C01814=1092.503,260.660,421.963,177.107,20.191,152.904
C01815=1092.509,260.908,421.935,177.110,20.194,152.904
C01816=1092.515,261.157,421.907,177.114,20.196,152.904
C01817=1092.520,261.405,421.880,177.117,20.198,152.904
C01818=1092.526,261.654,421.852,177.120,20.200,152.904
C01819=1092.533,261.902,421.825,177.122,20.202,152.904
C01820=1092.538,262.150,421.797,177.126,20.204,152.904
C01821=1092.547,262.515,421.756,177.131,20.208,152.904
C01822=1092.555,262.879,421.715,177.135,20.211,152.904
C01823=1092.563,263.243,421.675,177.139,20.215,152.904
C01824=1092.572,263.608,421.634,177.144,20.218,152.904
C01825=1092.577,263.856,421.606,177.147,20.220,152.903
C01826=1092.583,264.105,421.578,177.150,20.222,152.903
C01827=1092.589,264.353,421.550,177.153,20.224,152.903
C01828=1092.595,264.601,421.522,177.157,20.227,152.903
C01829=1092.601,264.849,421.494,177.159,20.229,152.903
C01830=1092.606,265.097,421.466,177.162,20.231,152.903
C01831=1092.612,265.346,421.438,177.165,20.233,152.903
C01832=1092.617,265.594,421.410,177.169,20.236,152.903
C01833=1092.623,265.843,421.381,177.172,20.239,152.903
C01834=1092.629,266.091,421.353,177.174,20.241,152.904
C01835=1092.635,266.340,421.325,177.177,20.243,152.903
C01836=1092.640,266.588,421.297,177.181,20.245,152.903
C01837=1092.645,266.836,421.269,177.184,20.248,152.903
C01838=1092.651,267.085,421.241,177.187,20.250,152.904
C01839=1092.656,267.333,421.213,177.189,20.252,152.903
C01840=1092.662,267.581,421.184,177.193,20.254,152.903
C01841=1092.668,267.829,421.157,177.196,20.257,152.904
C01842=1092.674,268.078,421.128,177.199,20.259,152.903
C01843=1092.679,268.326,421.100,177.202,20.261,152.903
C01844=1092.685,268.575,421.072,177.206,20.264,152.903
C01845=1092.690,268.823,421.044,177.208,20.266,152.904
C01846=1092.697,269.071,421.015,177.211,20.268,152.903
C01847=1092.702,269.319,420.987,177.214,20.271,152.903
C01848=1092.708,269.568,420.959,177.218,20.273,152.903
C01849=1092.714,269.817,420.930,177.221,20.276,152.904
C01850=1092.719,270.065,420.902,177.223,20.278,152.904
C01851=1092.725,270.313,420.873,177.226,20.280,152.903
C01852=1092.730,270.561,420.845,177.230,20.282,152.904
C01853=1092.736,270.810,420.816,177.233,20.285,152.904
C01854=1092.741,271.058,420.788,177.236,20.287,152.904
C01855=1092.748,271.306,420.759,177.239,20.290,152.904
C01856=1092.753,271.554,420.731,177.242,20.292,152.904
C01857=1092.759,271.803,420.703,177.245,20.294,152.904
C01858=1092.764,272.051,420.674,177.248,20.296,152.904
C01859=1092.770,272.300,420.646,177.251,20.299,152.904
C01860=1092.776,272.548,420.617,177.254,20.301,152.904
C01861=1092.781,272.796,420.589,177.257,20.304,152.904
C01862=1092.787,273.044,420.560,177.261,20.306,152.904
C01863=1092.792,273.293,420.532,177.263,20.308,152.904
C01864=1092.798,273.541,420.503,177.266,20.311,152.904
C01865=1092.804,273.790,420.474,177.269,20.313,152.904
C01866=1092.810,274.037,420.446,177.273,20.316,152.904
C01867=1092.815,274.286,420.417,177.276,20.318,152.904
C01868=1092.821,274.534,420.388,177.279,20.321,152.904
C01869=1092.826,274.782,420.360,177.282,20.323,152.904
C01870=1092.832,275.031,420.331,177.285,20.325,152.904
C01871=1092.837,275.279,420.302,177.288,20.327,152.904
C01872=1092.843,275.528,420.274,177.291,20.330,152.904
C01873=1092.852,275.895,420.231,177.296,20.333,152.904
C01874=1092.860,276.262,420.188,177.300,20.337,152.904
C01875=1092.868,276.628,420.146,177.304,20.340,152.904
C01876=1092.877,276.995,420.104,177.309,20.344,152.904
C01877=1092.882,277.244,420.074,177.313,20.346,152.904
C01878=1092.888,277.492,420.045,177.316,20.349,152.904
C01879=1092.894,277.740,420.017,177.319,20.352,152.904
C01880=1092.899,277.988,419.987,177.322,20.354,152.904
C01881=1092.905,278.237,419.958,177.325,20.357,152.904
C01882=1092.910,278.485,419.930,177.328,20.359,152.904
C01883=1092.916,278.733,419.901,177.331,20.361,152.904
C01884=1092.922,278.981,419.871,177.334,20.364,152.904
C01885=1092.927,279.230,419.843,177.337,20.366,152.904
C01886=1092.933,279.478,419.814,177.340,20.369,152.904
C01887=1092.939,279.726,419.784,177.343,20.371,152.905
C01888=1092.945,279.974,419.755,177.346,20.374,152.905
C01889=1092.950,280.223,419.727,177.350,20.376,152.905
C01890=1092.956,280.471,419.698,177.353,20.379,152.905
C01891=1092.962,280.719,419.668,177.356,20.381,152.905
C01892=1092.968,280.967,419.639,177.359,20.384,152.905
C01893=1092.973,281.215,419.610,177.361,20.386,152.905
C01894=1092.979,281.463,419.581,177.365,20.388,152.905
C01895=1092.984,281.712,419.552,177.368,20.391,152.905
C01896=1092.990,281.961,419.522,177.371,20.393,152.905
C01897=1092.995,282.208,419.494,177.374,20.396,152.905
C01898=1093.001,282.457,419.464,177.377,20.398,152.905
C01899=1093.007,282.705,419.435,177.380,20.401,152.905
C01900=1093.013,282.953,419.405,177.384,20.404,152.905
C01901=1093.017,283.201,419.376,177.387,20.407,152.905
C01902=1093.024,283.449,419.347,177.390,20.409,152.905
C01903=1093.029,283.697,419.317,177.393,20.412,152.905
C01904=1093.035,283.946,419.288,177.396,20.414,152.905
C01905=1093.040,284.193,419.259,177.399,20.417,152.905
C01906=1093.046,284.442,419.229,177.402,20.419,152.905
C01907=1093.051,284.690,419.200,177.405,20.421,152.906
C01908=1093.058,284.938,419.171,177.408,20.424,152.906
C01909=1093.063,285.187,419.141,177.411,20.426,152.906
C01910=1093.069,285.435,419.112,177.414,20.429,152.906
C01911=1093.074,285.683,419.083,177.417,20.432,152.906
C01912=1093.080,285.931,419.053,177.420,20.434,152.906
C01913=1093.085,286.180,419.024,177.424,20.437,152.906
C01914=1093.091,286.427,418.993,177.427,20.439,152.906
C01915=1093.097,286.675,418.964,177.430,20.442,152.906
C01916=1093.103,286.924,418.935,177.433,20.444,152.906
C01917=1093.108,287.172,418.905,177.436,20.447,152.906
C01918=1093.114,287.420,418.876,177.439,20.450,152.906
C01919=1093.120,287.668,418.847,177.442,20.452,152.906
C01920=1093.125,287.916,418.816,177.445,20.455,152.906
C01921=1093.131,288.164,418.787,177.449,20.457,152.906
C01922=1093.137,288.413,418.758,177.452,20.460,152.906
C01923=1093.143,288.661,418.728,177.455,20.462,152.907
C01924=1093.149,288.909,418.698,177.458,20.465,152.907
C01925=1093.157,289.285,418.653,177.463,20.469,152.907
C01926=1093.166,289.662,418.608,177.467,20.473,152.907
C01927=1093.174,290.038,418.562,177.472,20.477,152.907
C01928=1093.184,290.415,418.517,177.477,20.481,152.907
C01929=1093.188,290.663,418.488,177.480,20.484,152.907
C01930=1093.194,290.911,418.458,177.483,20.486,152.907
C01931=1093.200,291.159,418.428,177.486,20.489,152.907
C01932=1093.205,291.407,418.398,177.489,20.492,152.907
C01933=1093.211,291.655,418.368,177.492,20.494,152.907
C01934=1093.217,291.903,418.338,177.496,20.497,152.908
C01935=1093.222,292.151,418.308,177.498,20.500,152.908
C01936=1093.228,292.400,418.278,177.502,20.502,152.908
C01937=1093.234,292.648,418.248,177.505,20.505,152.908
C01938=1093.239,292.896,418.218,177.508,20.508,152.908
C01939=1093.245,293.144,418.188,177.511,20.510,152.908
C01940=1093.251,293.392,418.158,177.514,20.513,152.908
C01941=1093.256,293.640,418.128,177.517,20.516,152.908
C01942=1093.262,293.889,418.098,177.520,20.518,152.908
C01943=1093.268,294.136,418.068,177.523,20.521,152.908
C01944=1093.273,294.385,418.038,177.526,20.524,152.909
C01945=1093.279,294.633,418.008,177.530,20.526,152.909
C01946=1093.285,294.880,417.978,177.533,20.529,152.909
C01947=1093.290,295.129,417.948,177.536,20.532,152.909
C01948=1093.296,295.377,417.918,177.539,20.534,152.909
C01949=1093.302,295.625,417.887,177.542,20.537,152.909
C01950=1093.308,295.873,417.858,177.545,20.540,152.909
C01951=1093.313,296.121,417.827,177.548,20.542,152.909
C01952=1093.319,296.369,417.797,177.551,20.545,152.909
C01953=1093.325,296.616,417.767,177.554,20.548,152.909
C01954=1093.330,296.865,417.737,177.557,20.550,152.909
C01955=1093.336,297.113,417.706,177.560,20.553,152.910
C01956=1093.341,297.361,417.676,177.564,20.556,152.910
C01957=1093.348,297.609,417.645,177.567,20.559,152.910
C01958=1093.353,297.858,417.615,177.570,20.561,152.910
C01959=1093.359,298.106,417.585,177.573,20.564,152.910
C01960=1093.364,298.354,417.554,177.576,20.567,152.910
C01961=1093.370,298.602,417.524,177.579,20.570,152.910
C01962=1093.376,298.849,417.493,177.582,20.572,152.910
C01963=1093.381,299.098,417.462,177.585,20.575,152.911
C01964=1093.386,299.346,417.433,177.588,20.578,152.911
C01965=1093.392,299.594,417.402,177.592,20.581,152.911
C01966=1093.397,299.842,417.371,177.595,20.584,152.911
C01967=1093.403,300.090,417.341,177.598,20.587,152.911
C01968=1093.409,300.338,417.311,177.601,20.590,152.911
C01969=1093.414,300.586,417.280,177.604,20.593,152.911
C01970=1093.420,300.834,417.249,177.607,20.596,152.912
C01971=1093.425,301.082,417.218,177.610,20.598,152.912
C01972=1093.431,301.330,417.188,177.613,20.601,152.912
C01973=1093.437,301.578,417.157,177.616,20.604,152.912
C01974=1093.442,301.826,417.126,177.619,20.607,152.912
C01975=1093.448,302.074,417.096,177.622,20.609,152.912
C01976=1093.453,302.322,417.065,177.625,20.612,152.913
C01977=1093.463,302.712,417.017,177.631,20.617,152.913
C01978=1093.471,303.103,416.968,177.635,20.621,152.913
C01979=1093.480,303.493,416.920,177.640,20.626,152.913
C01980=1093.489,303.884,416.871,177.645,20.630,152.913
C01981=1093.495,304.131,416.841,177.648,20.633,152.914
C01982=1093.500,304.380,416.810,177.651,20.636,152.914
C01983=1093.506,304.627,416.779,177.655,20.639,152.914
C01984=1093.512,304.876,416.747,177.658,20.642,152.914
C01985=1093.517,305.123,416.717,177.661,20.645,152.914
C01986=1093.523,305.372,416.686,177.664,20.648,152.914
C01987=1093.528,305.619,416.656,177.667,20.651,152.914
C01988=1093.534,305.867,416.624,177.670,20.654,152.915
C01989=1093.540,306.115,416.593,177.673,20.657,152.915
C01990=1093.545,306.364,416.562,177.676,20.659,152.915
C01991=1093.551,306.611,416.531,177.679,20.662,152.915
C01992=1093.556,306.859,416.500,177.683,20.666,152.915
C01993=1093.563,307.107,416.470,177.686,20.669,152.915
C01994=1093.568,307.355,416.438,177.689,20.672,152.916
C01995=1093.574,307.603,416.408,177.692,20.674,152.916
C01996=1093.580,307.852,416.376,177.695,20.677,152.916
C01997=1093.586,308.099,416.345,177.698,20.680,152.916
C01998=1093.591,308.347,416.314,177.701,20.683,152.916
C01999=1093.597,308.594,416.283,177.705,20.686,152.916
C02000=1093.603,308.843,416.252,177.708,20.689,152.916
C02001=1093.608,309.090,416.220,177.711,20.692,152.917
C02002=1093.614,309.338,416.190,177.714,20.695,152.917
C02003=1093.620,309.586,416.158,177.717,20.698,152.917
C02004=1093.626,309.834,416.128,177.720,20.701,152.917
C02005=1093.632,310.083,416.096,177.723,20.703,152.917
C02006=1093.637,310.331,416.065,177.726,20.706,152.917
C02007=1093.643,310.578,416.034,177.730,20.710,152.918
C02008=1093.649,310.827,416.002,177.733,20.713,152.918
C02009=1093.655,311.074,415.971,177.735,20.716,152.918
C02010=1093.660,311.323,415.940,177.738,20.719,152.918
C02011=1093.666,311.570,415.908,177.742,20.721,152.918
C02012=1093.672,311.817,415.877,177.745,20.724,152.918
C02013=1093.678,312.066,415.846,177.748,20.728,152.919
C02014=1093.683,312.314,415.814,177.751,20.731,152.919
C02015=1093.690,312.562,415.783,177.754,20.734,152.919
C02016=1093.695,312.810,415.752,177.757,20.737,152.919
C02017=1093.701,313.058,415.720,177.760,20.740,152.919
C02018=1093.707,313.305,415.689,177.763,20.743,152.920
C02019=1093.713,313.554,415.657,177.766,20.746,152.920
C02020=1093.718,313.802,415.626,177.770,20.749,152.920
C02021=1093.724,314.050,415.594,177.773,20.751,152.920
C02022=1093.730,314.297,415.563,177.776,20.754,152.920
C02023=1093.736,314.546,415.531,177.779,20.757,152.920
C02024=1093.741,314.793,415.500,177.782,20.760,152.921
C02025=1093.748,315.041,415.468,177.786,20.764,152.921
C02026=1093.753,315.289,415.437,177.789,20.767,152.921
C02027=1093.759,315.537,415.405,177.792,20.770,152.921
C02028=1093.765,315.784,415.373,177.795,20.773,152.922
C02029=1093.773,316.178,415.322,177.800,20.778,152.922
C02030=1093.782,316.571,415.272,177.804,20.783,152.922
C02031=1093.791,316.964,415.222,177.809,20.788,152.923
C02032=1093.799,317.357,415.171,177.814,20.793,152.923
C02033=1093.805,317.605,415.139,177.817,20.797,152.923
C02034=1093.811,317.853,415.108,177.820,20.800,152.924
C02035=1093.817,318.101,415.076,177.823,20.803,152.924
C02036=1093.822,318.349,415.044,177.827,20.807,152.924
C02037=1093.828,318.597,415.012,177.830,20.810,152.924
C02038=1093.833,318.844,414.980,177.833,20.813,152.924
C02039=1093.839,319.093,414.948,177.835,20.816,152.925
C02040=1093.845,319.340,414.916,177.838,20.819,152.925
C02041=1093.850,319.589,414.884,177.842,20.822,152.925
C02042=1093.855,319.836,414.852,177.845,20.826,152.926
C02043=1093.861,320.084,414.820,177.848,20.829,152.926
C02044=1093.867,320.333,414.788,177.851,20.832,152.926
C02045=1093.873,320.579,414.756,177.855,20.836,152.926
C02046=1093.879,320.828,414.724,177.858,20.839,152.926
C02047=1093.884,321.075,414.691,177.860,20.842,152.927
C02048=1093.890,321.324,414.659,177.863,20.845,152.927
C02049=1093.895,321.571,414.628,177.867,20.849,152.927
C02050=1093.901,321.819,414.595,177.870,20.852,152.927
C02051=1093.907,322.067,414.563,177.873,20.855,152.928
C02052=1093.913,322.315,414.531,177.876,20.858,152.928
C02053=1093.918,322.563,414.499,177.879,20.862,152.928
C02054=1093.924,322.811,414.466,177.882,20.865,152.929
C02055=1093.930,323.058,414.434,177.885,20.868,152.929
C02056=1093.936,323.306,414.402,177.888,20.872,152.929
C02057=1093.941,323.555,414.370,177.892,20.875,152.929
C02058=1093.946,323.802,414.337,177.894,20.878,152.930
C02059=1093.952,324.050,414.305,177.897,20.881,152.930
C02060=1093.958,324.298,414.273,177.900,20.885,152.930
C02061=1093.963,324.545,414.240,177.904,20.888,152.930
C02062=1093.969,324.794,414.208,177.907,20.892,152.931
C02063=1093.976,325.041,414.176,177.910,20.895,152.931
C02064=1093.981,325.289,414.144,177.912,20.898,152.931
C02065=1093.986,325.537,414.111,177.916,20.902,152.932
C02066=1093.993,325.785,414.078,177.919,20.905,152.932
C02067=1093.999,326.033,414.046,177.922,20.908,152.932
C02068=1094.004,326.280,414.014,177.926,20.912,152.932
C02069=1094.010,326.528,413.981,177.928,20.915,152.933
C02070=1094.016,326.776,413.949,177.931,20.918,152.933
C02071=1094.022,327.024,413.917,177.934,20.921,152.933
C02072=1094.027,327.272,413.883,177.938,20.925,152.933
C02073=1094.033,327.519,413.851,177.941,20.928,152.934
C02074=1094.039,327.767,413.819,177.944,20.932,152.934
C02075=1094.045,328.015,413.786,177.947,20.936,152.934
C02076=1094.051,328.263,413.754,177.950,20.939,152.935
C02077=1094.057,328.511,413.721,177.953,20.942,152.935
C02078=1094.062,328.758,413.688,177.956,20.946,152.935
C02079=1094.068,329.006,413.656,177.959,20.949,152.935
C02080=1094.074,329.254,413.623,177.962,20.952,152.936
C02081=1094.083,329.640,413.572,177.967,20.958,152.936
C02082=1094.092,330.027,413.521,177.972,20.963,152.937
C02083=1094.101,330.413,413.470,177.977,20.969,152.937
C02084=1094.110,330.799,413.419,177.982,20.974,152.938
C02085=1094.116,331.046,413.386,177.985,20.978,152.938
C02086=1094.122,331.295,413.354,177.988,20.981,152.938
C02087=1094.128,331.543,413.320,177.991,20.984,152.939
C02088=1094.134,331.790,413.288,177.995,20.988,152.939
C02089=1094.140,332.038,413.254,177.997,20.991,152.939
C02090=1094.145,332.285,413.222,178.000,20.995,152.940
C02091=1094.151,332.533,413.189,178.004,20.999,152.940
C02092=1094.156,332.781,413.155,178.006,21.002,152.940
C02093=1094.162,333.029,413.123,178.009,21.005,152.941
C02094=1094.168,333.277,413.090,178.013,21.009,152.941
C02095=1094.173,333.525,413.057,178.016,21.013,152.941
C02096=1094.180,333.772,413.024,178.019,21.017,152.942
C02097=1094.185,334.020,412.991,178.022,21.020,152.942
C02098=1094.190,334.267,412.958,178.025,21.023,152.942
C02099=1094.197,334.515,412.925,178.028,21.027,152.943
C02100=1094.202,334.763,412.891,178.031,21.031,152.943
C02101=1094.208,335.011,412.858,178.035,21.035,152.943
C02102=1094.213,335.259,412.825,178.037,21.039,152.944
C02103=1094.220,335.506,412.792,178.040,21.042,152.944
C02104=1094.225,335.754,412.759,178.044,21.046,152.944
C02105=1094.231,336.002,412.725,178.047,21.049,152.945
C02106=1094.237,336.249,412.692,178.050,21.053,152.945
C02107=1094.243,336.497,412.659,178.053,21.057,152.945
C02108=1094.248,336.745,412.625,178.055,21.060,152.946
C02109=1094.254,336.993,412.592,178.059,21.064,152.946
C02110=1094.260,337.240,412.559,178.062,21.068,152.947
C02111=1094.266,337.488,412.526,178.066,21.072,152.947
C02112=1094.272,337.736,412.492,178.068,21.075,152.947
C02113=1094.277,337.984,412.458,178.071,21.079,152.948
C02114=1094.283,338.231,412.425,178.074,21.083,152.948
C02115=1094.289,338.479,412.392,178.077,21.086,152.948
C02116=1094.295,338.727,412.359,178.081,21.090,152.949
C02117=1094.300,338.974,412.325,178.083,21.094,152.949
C02118=1094.306,339.222,412.292,178.087,21.098,152.950
C02119=1094.312,339.470,412.258,178.090,21.102,152.950
C02120=1094.317,339.717,412.224,178.093,21.105,152.950
C02121=1094.323,339.965,412.191,178.096,21.109,152.951
C02122=1094.329,340.213,412.158,178.099,21.113,152.951
C02123=1094.334,340.460,412.124,178.102,21.117,152.952
C02124=1094.340,340.708,412.090,178.105,21.120,152.952
C02125=1094.346,340.956,412.056,178.108,21.125,152.953
C02126=1094.351,341.204,412.023,178.111,21.128,152.953
C02127=1094.357,341.451,411.989,178.114,21.133,152.953
C02128=1094.363,341.699,411.955,178.117,21.136,152.954
C02129=1094.368,341.947,411.922,178.121,21.140,152.954
C02130=1094.375,342.195,411.888,178.123,21.144,152.955
C02131=1094.380,342.443,411.854,178.127,21.148,152.955
C02132=1094.386,342.690,411.820,178.129,21.152,152.955
C02133=1094.395,343.070,411.769,178.134,21.158,152.956
C02134=1094.404,343.450,411.717,178.139,21.164,152.957
C02135=1094.413,343.830,411.664,178.144,21.170,152.957
C02136=1094.421,344.210,411.613,178.149,21.176,152.958
C02137=1094.428,344.458,411.579,178.151,21.179,152.958
C02138=1094.433,344.706,411.546,178.155,21.184,152.959
C02139=1094.439,344.953,411.511,178.157,21.187,152.959
C02140=1094.445,345.200,411.477,178.161,21.192,152.960
C02141=1094.450,345.449,411.444,178.163,21.196,152.960
C02142=1094.456,345.696,411.409,178.167,21.200,152.961
C02143=1094.462,345.944,411.375,178.170,21.203,152.961
C02144=1094.468,346.191,411.341,178.173,21.208,152.962
C02145=1094.474,346.439,411.308,178.176,21.212,152.962
C02146=1094.479,346.687,411.273,178.179,21.216,152.963
C02147=1094.485,346.934,411.239,178.183,21.220,152.963
C02148=1094.491,347.181,411.205,178.185,21.224,152.964
C02149=1094.497,347.429,411.170,178.189,21.228,152.964
C02150=1094.502,347.677,411.137,178.191,21.232,152.965
C02151=1094.508,347.925,411.102,178.195,21.237,152.965
C02152=1094.514,348.172,411.068,178.197,21.240,152.965
C02153=1094.520,348.420,411.034,178.201,21.245,152.966
C02154=1094.525,348.668,410.999,178.203,21.249,152.966
C02155=1094.531,348.915,410.965,178.207,21.253,152.967
C02156=1094.537,349.162,410.931,178.210,21.257,152.967
C02157=1094.542,349.410,410.897,178.213,21.261,152.968
C02158=1094.549,349.658,410.862,178.216,21.265,152.968
C02159=1094.554,349.905,410.828,178.219,21.269,152.969
C02160=1094.559,350.153,410.793,178.222,21.274,152.969
C02161=1094.566,350.401,410.759,178.224,21.278,152.970
C02162=1094.572,350.648,410.725,178.228,21.282,152.970
C02163=1094.577,350.896,410.690,178.231,21.286,152.971
C02164=1094.583,351.143,410.656,178.234,21.290,152.971
C02165=1094.589,351.391,410.622,178.237,21.295,152.972
C02166=1094.594,351.638,410.587,178.240,21.299,152.972
C02167=1094.600,351.886,410.553,178.243,21.303,152.973
C02168=1094.606,352.133,410.517,178.247,21.308,152.973
C02169=1094.612,352.381,410.483,178.249,21.311,152.974
C02170=1094.618,352.628,410.449,178.252,21.316,152.975
C02171=1094.624,352.876,410.414,178.255,21.320,152.975
C02172=1094.630,353.123,410.380,178.258,21.324,152.976
C02173=1094.635,353.370,410.345,178.262,21.329,152.976
C02174=1094.641,353.618,410.311,178.264,21.333,152.977
C02175=1094.647,353.866,410.276,178.268,21.338,152.977
C02176=1094.652,354.113,410.242,178.271,21.342,152.978
C02177=1094.658,354.361,410.206,178.273,21.346,152.978
C02178=1094.664,354.608,410.172,178.277,21.351,152.979
C02179=1094.669,354.856,410.137,178.279,21.355,152.979
C02180=1094.675,355.104,410.102,178.283,21.359,152.980
C02181=1094.681,355.351,410.068,178.286,21.364,152.981
C02182=1094.686,355.598,410.033,178.288,21.368,152.981
C02183=1094.693,355.846,409.998,178.292,21.372,152.982
C02184=1094.698,356.093,409.963,178.295,21.377,152.982
C02185=1094.708,356.476,409.909,178.299,21.384,152.983
C02186=1094.716,356.858,409.855,178.304,21.391,152.984
C02187=1094.726,357.242,409.801,178.308,21.398,152.985
C02188=1094.734,357.624,409.747,178.314,21.405,152.986
C02189=1094.740,357.871,409.712,178.316,21.409,152.986
C02190=1094.745,358.119,409.677,178.319,21.414,152.987
C02191=1094.752,358.366,409.642,178.323,21.418,152.988
C02192=1094.758,358.614,409.607,178.325,21.422,152.988
C02193=1094.763,358.861,409.572,178.328,21.427,152.989
C02194=1094.770,359.108,409.537,178.332,21.432,152.989
C02195=1094.775,359.356,409.502,178.334,21.436,152.990
C02196=1094.781,359.604,409.466,178.337,21.441,152.991
C02197=1094.787,359.850,409.432,178.341,21.446,152.991
C02198=1094.793,360.099,409.397,178.344,21.450,152.992
C02199=1094.798,360.346,409.361,178.346,21.454,152.992
C02200=1094.804,360.593,409.326,178.350,21.459,152.993
C02201=1094.810,360.840,409.291,178.353,21.464,152.994
C02202=1094.816,361.088,409.256,178.355,21.468,152.994
C02203=1094.821,361.335,409.220,178.358,21.473,152.995
C02204=1094.827,361.583,409.185,178.362,21.478,152.996
C02205=1094.833,361.830,409.149,178.365,21.483,152.996
C02206=1094.839,362.078,409.114,178.367,21.487,152.997
C02207=1094.845,362.325,409.080,178.371,21.492,152.998
C02208=1094.851,362.573,409.044,178.374,21.497,152.998
C02209=1094.856,362.820,409.008,178.377,21.502,152.999
C02210=1094.862,363.067,408.973,178.379,21.506,153.000
C02211=1094.868,363.315,408.937,178.383,21.511,153.000
C02212=1094.874,363.562,408.902,178.386,21.516,153.001
C02213=1094.880,363.810,408.866,178.389,21.521,153.002
C02214=1094.885,364.057,408.831,178.391,21.525,153.002
C02215=1094.891,364.304,408.795,178.394,21.530,153.003
C02216=1094.897,364.551,408.759,178.398,21.535,153.004
C02217=1094.903,364.799,408.724,178.401,21.540,153.004
C02218=1094.909,365.046,408.689,178.403,21.544,153.005
C02219=1094.915,365.293,408.653,178.406,21.549,153.006
C02220=1094.921,365.541,408.617,178.409,21.554,153.006
C02221=1094.926,365.788,408.582,178.413,21.559,153.007
C02222=1094.932,366.035,408.546,178.416,21.564,153.008
C02223=1094.938,366.283,408.511,178.418,21.569,153.008
C02224=1094.943,366.530,408.475,178.421,21.574,153.009
C02225=1094.949,366.778,408.438,178.424,21.579,153.010
C02226=1094.955,367.024,408.403,178.427,21.584,153.011
C02227=1094.961,367.272,408.367,178.431,21.589,153.011
C02228=1094.967,367.520,408.331,178.433,21.593,153.012
C02229=1094.972,367.767,408.296,178.436,21.599,153.013
C02230=1094.979,368.014,408.260,178.439,21.604,153.013
C02231=1094.984,368.262,408.223,178.442,21.609,153.014
C02232=1094.989,368.509,408.188,178.445,21.614,153.015
C02233=1094.995,368.756,408.152,178.448,21.619,153.016
C02234=1095.001,369.003,408.116,178.451,21.623,153.016
C02235=1095.007,369.251,408.080,178.454,21.629,153.017
C02236=1095.013,369.498,408.045,178.457,21.634,153.018
C02237=1095.022,369.896,407.986,178.462,21.642,153.019
C02238=1095.032,370.294,407.928,178.467,21.650,153.020
C02239=1095.041,370.691,407.870,178.471,21.658,153.022
C02240=1095.050,371.089,407.813,178.475,21.667,153.023
C02241=1095.057,371.337,407.776,178.479,21.672,153.024
C02242=1095.061,371.584,407.740,178.482,21.677,153.024
C02243=1095.068,371.831,407.704,178.485,21.682,153.025
C02244=1095.074,372.079,407.668,178.488,21.687,153.026
C02245=1095.080,372.326,407.632,178.491,21.693,153.027
C02246=1095.085,372.572,407.595,178.494,21.698,153.028
C02247=1095.091,372.820,407.559,178.496,21.703,153.028
C02248=1095.097,373.067,407.523,178.499,21.708,153.029
C02249=1095.104,373.315,407.487,178.502,21.713,153.030
C02250=1095.109,373.562,407.450,178.505,21.719,153.031
C02251=1095.115,373.808,407.414,178.508,21.724,153.031
C02252=1095.121,374.056,407.378,178.511,21.729,153.032
C02253=1095.126,374.303,407.341,178.514,21.735,153.033
C02254=1095.133,374.550,407.305,178.517,21.740,153.034
C02255=1095.139,374.798,407.268,178.520,21.746,153.035
C02256=1095.144,375.045,407.232,178.523,21.751,153.036
C02257=1095.150,375.292,407.196,178.526,21.756,153.036
C02258=1095.156,375.539,407.159,178.528,21.761,153.037
C02259=1095.162,375.786,407.122,178.531,21.767,153.038
C02260=1095.167,376.034,407.086,178.534,21.772,153.039
C02261=1095.173,376.281,407.050,178.537,21.778,153.040
C02262=1095.179,376.528,407.013,178.540,21.783,153.041
C02263=1095.185,376.775,406.976,178.543,21.789,153.042
C02264=1095.191,377.022,406.939,178.546,21.794,153.042
C02265=1095.196,377.270,406.902,178.549,21.800,153.043
C02266=1095.203,377.517,406.866,178.552,21.805,153.044
C02267=1095.208,377.763,406.829,178.555,21.811,153.045
C02268=1095.214,378.011,406.793,178.557,21.817,153.046
C02269=1095.220,378.258,406.756,178.560,21.822,153.047
C02270=1095.226,378.505,406.719,178.563,21.828,153.048
C02271=1095.231,378.752,406.682,178.566,21.833,153.049
C02272=1095.237,379.000,406.645,178.569,21.839,153.050
C02273=1095.243,379.247,406.609,178.572,21.845,153.051
C02274=1095.249,379.494,406.572,178.575,21.850,153.051
C02275=1095.255,379.741,406.535,178.578,21.856,153.052
C02276=1095.261,379.988,406.498,178.581,21.861,153.053
C02277=1095.267,380.236,406.462,178.584,21.867,153.054
C02278=1095.272,380.482,406.425,178.587,21.873,153.055
C02279=1095.278,380.729,406.387,178.589,21.879,153.056
C02280=1095.285,380.976,406.351,178.592,21.884,153.057
C02281=1095.290,381.223,406.314,178.595,21.890,153.058
C02282=1095.296,381.471,406.277,178.598,21.895,153.059
C02283=1095.302,381.718,406.240,178.601,21.901,153.060
C02284=1095.308,381.965,406.203,178.604,21.907,153.061
C02285=1095.314,382.212,406.166,178.607,21.913,153.062
C02286=1095.320,382.459,406.129,178.609,21.919,153.063
C02287=1095.326,382.706,406.091,178.612,21.924,153.064
C02288=1095.331,382.953,406.054,178.615,21.930,153.065
C02289=1095.337,383.165,406.023,178.618,21.935,153.065
C02290=1095.341,383.378,405.990,178.620,21.940,153.066
C02291=1095.347,383.591,405.959,178.623,21.946,153.067
C02292=1095.351,383.803,405.926,178.625,21.951,153.068
C02293=1095.356,384.016,405.895,178.627,21.956,153.069
C02294=1095.362,384.229,405.862,178.630,21.961,153.070
C02295=1095.367,384.442,405.830,178.632,21.966,153.071
C02296=1095.372,384.654,405.797,178.635,21.971,153.071
C02297=1095.377,384.901,405.760,178.638,21.977,153.072
C02298=1095.383,385.148,405.723,178.641,21.984,153.073
C02299=1095.390,385.395,405.686,178.644,21.990,153.075
C02300=1095.396,385.642,405.648,178.646,21.996,153.076
C02301=1095.401,385.889,405.611,178.649,22.002,153.077
C02302=1095.407,386.136,405.574,178.652,22.008,153.078
C02303=1095.413,386.383,405.537,178.655,22.014,153.079
C02304=1095.419,386.630,405.499,178.657,22.020,153.080
C02305=1095.424,386.877,405.461,178.661,22.026,153.081
C02306=1095.430,387.124,405.424,178.664,22.032,153.082
C02307=1095.436,387.371,405.386,178.667,22.038,153.083
C02308=1095.442,387.618,405.349,178.669,22.045,153.084
C02309=1095.448,387.866,405.311,178.672,22.051,153.085
C02310=1095.454,388.112,405.273,178.675,22.057,153.086
C02311=1095.460,388.359,405.236,178.677,22.063,153.087
C02312=1095.465,388.607,405.199,178.681,22.070,153.088
C02313=1095.471,388.853,405.161,178.684,22.076,153.089
C02314=1095.477,389.100,405.123,178.686,22.082,153.090
C02315=1095.483,389.347,405.085,178.689,22.088,153.091
C02316=1095.490,389.594,405.047,178.692,22.094,153.093
C02317=1095.496,389.841,405.009,178.695,22.101,153.094
C02318=1095.501,390.088,404.972,178.698,22.107,153.095
C02319=1095.507,390.335,404.935,178.700,22.113,153.096
C02320=1095.513,390.582,404.897,178.703,22.119,153.097
C02321=1095.520,390.829,404.859,178.706,22.126,153.098
C02322=1095.525,391.076,404.821,178.709,22.133,153.099
C02323=1095.531,391.323,404.783,178.712,22.139,153.100
C02324=1095.537,391.569,404.745,178.714,22.145,153.101
C02325=1095.544,391.817,404.707,178.717,22.152,153.103
C02326=1095.549,392.064,404.669,178.720,22.158,153.104
C02327=1095.555,392.311,404.631,178.723,22.165,153.105
C02328=1095.561,392.557,404.593,178.726,22.171,153.106
C02329=1095.567,392.805,404.555,178.728,22.177,153.107
C02330=1095.572,393.052,404.517,178.731,22.184,153.108
C02331=1095.578,393.299,404.479,178.734,22.191,153.110
C02332=1095.585,393.546,404.441,178.737,22.198,153.111
C02333=1095.591,393.793,404.403,178.739,22.204,153.112
C02334=1095.596,394.039,404.364,178.742,22.210,153.113
C02335=1095.602,394.286,404.327,178.745,22.217,153.114
C02336=1095.609,394.533,404.288,178.748,22.224,153.116
C02337=1095.614,394.781,404.250,178.750,22.231,153.117
C02338=1095.620,395.027,404.212,178.754,22.238,153.118
C02339=1095.626,395.274,404.173,178.756,22.244,153.119
C02340=1095.632,395.521,404.135,178.759,22.251,153.120
C02341=1095.638,395.769,404.097,178.761,22.257,153.122
C02342=1095.644,396.015,404.059,178.765,22.265,153.123
C02343=1095.650,396.262,404.020,178.767,22.271,153.124
C02344=1095.656,396.509,403.982,178.770,22.278,153.125
C02345=1095.661,396.728,403.948,178.772,22.284,153.127
C02346=1095.667,396.947,403.914,178.775,22.290,153.128
C02347=1095.671,397.166,403.880,178.777,22.296,153.129
C02348=1095.677,397.385,403.846,178.780,22.303,153.130
C02349=1095.682,397.604,403.812,178.782,22.309,153.131
C02350=1095.687,397.823,403.777,178.785,22.315,153.132
C02351=1095.692,398.042,403.744,178.787,22.321,153.133
C02352=1095.698,398.261,403.709,178.789,22.327,153.135
C02353=1095.704,398.507,403.670,178.793,22.335,153.136
C02354=1095.710,398.755,403.632,178.795,22.342,153.137
C02355=1095.716,399.001,403.593,178.797,22.348,153.138
C02356=1095.722,399.249,403.554,178.801,22.356,153.140
C02357=1095.728,399.495,403.516,178.803,22.363,153.141
C02358=1095.733,399.743,403.477,178.806,22.369,153.142
C02359=1095.739,399.989,403.438,178.809,22.377,153.144
C02360=1095.745,400.237,403.400,178.811,22.384,153.145
C02361=1095.751,400.483,403.361,178.814,22.391,153.146
C02362=1095.757,400.730,403.322,178.817,22.399,153.148
C02363=1095.763,400.977,403.284,178.819,22.405,153.149
C02364=1095.769,401.224,403.244,178.822,22.413,153.150
C02365=1095.774,401.471,403.205,178.825,22.420,153.152
C02366=1095.781,401.718,403.167,178.828,22.428,153.153
C02367=1095.786,401.964,403.128,178.830,22.435,153.155
C02368=1095.793,402.212,403.089,178.833,22.442,153.156
C02369=1095.799,402.458,403.050,178.836,22.449,153.157
C02370=1095.805,402.705,403.011,178.839,22.457,153.159
C02371=1095.811,402.953,402.972,178.841,22.464,153.160
C02372=1095.816,403.199,402.933,178.844,22.472,153.162
C02373=1095.823,403.446,402.894,178.847,22.479,153.163
C02374=1095.828,403.692,402.855,178.850,22.487,153.165
C02375=1095.834,403.939,402.816,178.852,22.494,153.166
C02376=1095.840,404.187,402.776,178.855,22.502,153.167
C02377=1095.847,404.433,402.738,178.857,22.509,153.169
C02378=1095.853,404.680,402.698,178.861,22.517,153.170
C02379=1095.858,404.926,402.659,178.863,22.524,153.172
C02380=1095.864,405.173,402.620,178.866,22.532,153.173
C02381=1095.870,405.420,402.580,178.868,22.539,153.175
C02382=1095.876,405.667,402.541,178.871,22.547,153.176
C02383=1095.883,405.914,402.502,178.874,22.555,153.178
C02384=1095.889,406.161,402.463,178.877,22.563,153.179
C02385=1095.894,406.407,402.424,178.880,22.571,153.181
C02386=1095.900,406.654,402.385,178.882,22.578,153.182
C02387=1095.906,406.902,402.345,178.885,22.586,153.184
C02388=1095.912,407.148,402.306,178.887,22.594,153.185
C02389=1095.918,407.395,402.266,178.890,22.602,153.187
C02390=1095.924,407.642,402.226,178.893,22.610,153.188
C02391=1095.930,407.889,402.187,178.895,22.617,153.190
C02392=1095.936,408.135,402.148,178.898,22.626,153.191
C02393=1095.942,408.382,402.109,178.901,22.633,153.193
C02394=1095.948,408.629,402.068,178.904,22.641,153.194
C02395=1095.953,408.876,402.029,178.907,22.650,153.196
C02396=1095.959,409.123,401.989,178.909,22.657,153.198
C02397=1095.965,409.369,401.949,178.912,22.665,153.199
C02398=1095.972,409.616,401.910,178.914,22.674,153.201
C02399=1095.977,409.862,401.870,178.917,22.682,153.202
C02400=1095.983,410.109,401.831,178.920,22.690,153.204
C02401=1095.989,410.329,401.796,178.922,22.697,153.205
C02402=1095.994,410.548,401.759,178.924,22.704,153.207
C02403=1096.000,410.767,401.724,178.927,22.711,153.208
C02404=1096.005,410.987,401.689,178.930,22.719,153.210
C02405=1096.010,411.206,401.653,178.932,22.726,153.211
C02406=1096.015,411.425,401.619,178.934,22.734,153.213
C02407=1096.020,411.645,401.583,178.937,22.741,153.214
C02408=1096.026,411.864,401.547,178.939,22.749,153.216
C02409=1096.032,412.111,401.508,178.942,22.757,153.217
C02410=1096.038,412.357,401.468,178.945,22.765,153.219
C02411=1096.044,412.603,401.428,178.947,22.773,153.221
C02412=1096.050,412.851,401.388,178.950,22.782,153.222
C02413=1096.056,413.097,401.348,178.953,22.790,153.224
C02414=1096.062,413.344,401.307,178.955,22.799,153.226
C02415=1096.068,413.591,401.268,178.957,22.807,153.227
C02416=1096.074,413.838,401.227,178.960,22.816,153.229
C02417=1096.080,414.084,401.187,178.963,22.824,153.231
C02418=1096.087,414.331,401.147,178.966,22.833,153.233
C02419=1096.093,414.578,401.108,178.969,22.842,153.234
C02420=1096.098,414.825,401.067,178.972,22.850,153.236
C02421=1096.104,415.070,401.027,178.974,22.859,153.238
C02422=1096.111,415.317,400.987,178.976,22.868,153.240
C02423=1096.116,415.564,400.946,178.979,22.876,153.241
C02424=1096.123,415.810,400.906,178.982,22.885,153.243
C02425=1096.129,416.057,400.866,178.985,22.894,153.245
C02426=1096.135,416.304,400.825,178.987,22.903,153.247
C02427=1096.141,416.550,400.785,178.990,22.911,153.248
C02428=1096.147,416.797,400.745,178.993,22.920,153.250
C02429=1096.153,417.043,400.704,178.996,22.929,153.252
C02430=1096.159,417.290,400.664,178.998,22.938,153.254
C02431=1096.165,417.537,400.623,179.001,22.947,153.256
C02432=1096.171,417.784,400.582,179.004,22.956,153.258
C02433=1096.177,418.030,400.542,179.006,22.966,153.259
C02434=1096.183,418.277,400.502,179.008,22.974,153.261
C02435=1096.189,418.523,400.461,179.011,22.983,153.263
C02436=1096.195,418.770,400.421,179.014,22.992,153.265
C02437=1096.201,419.017,400.381,179.016,23.001,153.267
C02438=1096.207,419.263,400.339,179.019,23.010,153.269
C02439=1096.213,419.509,400.299,179.022,23.020,153.271
C02440=1096.219,419.756,400.258,179.024,23.029,153.273
C02441=1096.225,420.003,400.217,179.028,23.039,153.275
C02442=1096.232,420.250,400.176,179.030,23.048,153.276
C02443=1096.238,420.497,400.135,179.033,23.057,153.278
C02444=1096.244,420.743,400.095,179.036,23.066,153.280
C02445=1096.250,420.989,400.054,179.038,23.076,153.282
C02446=1096.256,421.236,400.013,179.041,23.085,153.284
C02447=1096.262,421.482,399.972,179.044,23.095,153.286
C02448=1096.268,421.729,399.932,179.046,23.104,153.288
C02449=1096.274,421.976,399.891,179.049,23.113,153.290
C02450=1096.280,422.222,399.850,179.051,23.123,153.292
C02451=1096.287,422.469,399.809,179.054,23.133,153.294
C02452=1096.293,422.715,399.767,179.056,23.142,153.296
C02453=1096.299,422.961,399.726,179.060,23.152,153.298
C02454=1096.305,423.208,399.686,179.062,23.162,153.300
C02455=1096.311,423.454,399.644,179.065,23.171,153.302
C02456=1096.316,423.701,399.604,179.067,23.181,153.304
C02457=1096.322,423.928,399.565,179.070,23.190,153.306
C02458=1096.328,424.154,399.527,179.072,23.199,153.308
C02459=1096.334,424.379,399.490,179.075,23.208,153.310
C02460=1096.339,424.606,399.453,179.077,23.217,153.312
C02461=1096.345,424.833,399.414,179.079,23.226,153.314
C02462=1096.350,425.059,399.376,179.082,23.235,153.316
C02463=1096.356,425.286,399.338,179.084,23.245,153.318
C02464=1096.361,425.512,399.300,179.086,23.254,153.320
C02465=1096.367,425.758,399.258,179.090,23.264,153.322
C02466=1096.373,426.005,399.218,179.092,23.274,153.324
C02467=1096.380,426.251,399.176,179.094,23.284,153.326
C02468=1096.386,426.498,399.134,179.097,23.294,153.328
C02469=1096.392,426.744,399.094,179.100,23.304,153.330
C02470=1096.398,426.990,399.052,179.102,23.315,153.333
C02471=1096.405,427.237,399.010,179.105,23.324,153.335
C02472=1096.411,427.483,398.969,179.107,23.335,153.337
C02473=1096.417,427.729,398.927,179.110,23.345,153.339
C02474=1096.423,427.976,398.886,179.113,23.355,153.341
C02475=1096.429,428.222,398.844,179.115,23.366,153.344
C02476=1096.435,428.468,398.803,179.118,23.376,153.346
C02477=1096.442,428.715,398.761,179.121,23.387,153.348
C02478=1096.448,428.962,398.719,179.123,23.397,153.350
C02479=1096.454,429.207,398.677,179.126,23.408,153.353
C02480=1096.460,429.454,398.635,179.128,23.418,153.355
C02481=1096.466,429.701,398.593,179.131,23.429,153.357
C02482=1096.472,429.947,398.552,179.134,23.439,153.359
C02483=1096.478,430.194,398.510,179.136,23.450,153.362
C02484=1096.484,430.439,398.468,179.138,23.461,153.364
C02485=1096.490,430.685,398.426,179.141,23.472,153.366
C02486=1096.497,430.932,398.385,179.144,23.482,153.369
C02487=1096.502,431.178,398.342,179.147,23.493,153.371
C02488=1096.508,431.424,398.300,179.149,23.504,153.373
C02489=1096.515,431.671,398.258,179.152,23.515,153.376
C02490=1096.521,431.917,398.216,179.154,23.526,153.378
C02491=1096.528,432.164,398.174,179.157,23.537,153.381
C02492=1096.533,432.410,398.132,179.159,23.548,153.383
C02493=1096.540,432.657,398.090,179.162,23.559,153.385
C02494=1096.546,432.902,398.048,179.165,23.570,153.388
C02495=1096.553,433.149,398.006,179.167,23.581,153.390
C02496=1096.558,433.395,397.963,179.170,23.592,153.393
C02497=1096.564,433.641,397.921,179.172,23.603,153.395
C02498=1096.571,433.887,397.879,179.175,23.615,153.398
C02499=1096.576,434.133,397.836,179.177,23.626,153.400
C02500=1096.583,434.380,397.795,179.180,23.637,153.403
C02501=1096.588,434.626,397.752,179.182,23.649,153.405
C02502=1096.595,434.872,397.709,179.185,23.660,153.408
C02503=1096.601,435.118,397.666,179.187,23.671,153.410
C02504=1096.607,435.365,397.625,179.190,23.683,153.413
C02505=1096.613,435.611,397.582,179.193,23.695,153.415
C02506=1096.620,435.857,397.539,179.195,23.706,153.418
C02507=1096.626,436.103,397.497,179.198,23.718,153.420
C02508=1096.632,436.350,397.454,179.200,23.730,153.423
C02509=1096.638,436.595,397.412,179.203,23.742,153.426
C02510=1096.645,436.842,397.369,179.205,23.753,153.428
C02511=1096.651,437.087,397.327,179.208,23.765,153.431
C02512=1096.657,437.334,397.283,179.210,23.777,153.433
C02513=1096.664,437.607,397.237,179.213,23.790,153.436
C02514=1096.670,437.881,397.189,179.215,23.803,153.439
C02515=1096.677,438.154,397.142,179.219,23.817,153.442
C02516=1096.685,438.428,397.093,179.221,23.830,153.445
C02517=1096.691,438.674,397.051,179.224,23.842,153.448
C02518=1096.697,438.920,397.008,179.227,23.854,153.451
C02519=1096.703,439.166,396.966,179.229,23.866,153.453
C02520=1096.709,439.412,396.923,179.231,23.878,153.456
C02521=1096.717,439.658,396.879,179.234,23.891,153.459
C02522=1096.723,439.905,396.836,179.236,23.903,153.462
C02523=1096.728,440.150,396.794,179.239,23.915,153.464
C02524=1096.735,440.397,396.751,179.242,23.927,153.467
C02525=1096.741,440.643,396.707,179.244,23.940,153.470
C02526=1096.747,440.889,396.664,179.246,23.952,153.473
C02527=1096.753,441.135,396.621,179.249,23.965,153.476
C02528=1096.760,441.381,396.578,179.251,23.978,153.478
C02529=1096.766,441.627,396.535,179.254,23.990,153.481
C02530=1096.772,441.873,396.491,179.256,24.003,153.484
C02531=1096.778,442.119,396.448,179.259,24.015,153.487
C02532=1096.785,442.365,396.404,179.261,24.028,153.490
C02533=1096.791,442.611,396.362,179.264,24.041,153.493
C02534=1096.797,442.857,396.318,179.266,24.054,153.496
C02535=1096.804,443.103,396.275,179.269,24.067,153.499
C02536=1096.810,443.349,396.231,179.271,24.080,153.502
C02537=1096.816,443.595,396.188,179.273,24.093,153.505
C02538=1096.822,443.841,396.144,179.276,24.106,153.508
C02539=1096.828,444.087,396.101,179.278,24.119,153.511
C02540=1096.835,444.333,396.057,179.280,24.132,153.514
C02541=1096.841,444.579,396.013,179.283,24.145,153.517
C02542=1096.848,444.825,395.970,179.284,24.158,153.520
C02543=1096.854,445.071,395.927,179.286,24.171,153.523
C02544=1096.860,445.317,395.883,179.287,24.184,153.526
C02545=1096.867,445.563,395.840,179.288,24.197,153.529
C02546=1096.873,445.809,395.796,179.289,24.210,153.532
C02547=1096.880,446.055,395.752,179.290,24.223,153.535
C02548=1096.885,446.301,395.707,179.292,24.236,153.539
C02549=1096.891,446.548,395.664,179.292,24.249,153.542
C02550=1096.898,446.794,395.620,179.293,24.262,153.545
C02551=1096.904,447.040,395.577,179.292,24.275,153.548
C02552=1096.911,447.285,395.533,179.293,24.288,153.551
C02553=1096.916,447.531,395.489,179.294,24.300,153.555
C02554=1096.923,447.777,395.445,179.293,24.313,153.558
C02555=1096.929,448.023,395.402,179.293,24.326,153.561
C02556=1096.936,448.269,395.358,179.293,24.339,153.564
C02557=1096.941,448.515,395.313,179.292,24.351,153.568
C02558=1096.948,448.761,395.269,179.292,24.365,153.571
C02559=1096.954,449.007,395.226,179.291,24.377,153.574
C02560=1096.961,449.252,395.181,179.291,24.390,153.578
C02561=1096.967,449.498,395.137,179.290,24.403,153.581
C02562=1096.974,449.744,395.093,179.289,24.416,153.584
C02563=1096.980,449.990,395.049,179.288,24.428,153.588
C02564=1096.988,450.237,395.006,179.287,24.440,153.591
C02565=1096.595,450.228,394.844,179.229,24.654,153.653
C02566=1096.588,449.983,394.887,179.230,24.642,153.649
C02567=1096.582,449.737,394.931,179.230,24.629,153.646
C02568=1096.575,449.491,394.976,179.232,24.616,153.643
C02569=1096.568,449.245,395.020,179.233,24.604,153.639
C02570=1096.562,448.999,395.063,179.233,24.590,153.636
C02571=1096.556,448.753,395.107,179.233,24.578,153.633
C02572=1096.550,448.508,395.152,179.234,24.565,153.629
C02573=1096.543,448.262,395.196,179.234,24.552,153.626
C02574=1096.537,448.016,395.240,179.234,24.539,153.623
C02575=1096.530,447.770,395.284,179.235,24.526,153.619
C02576=1096.524,447.524,395.328,179.235,24.513,153.616
C02577=1096.517,447.278,395.372,179.234,24.500,153.613
C02578=1096.511,447.032,395.416,179.234,24.488,153.610
C02579=1096.505,446.786,395.460,179.234,24.475,153.606
C02580=1096.499,446.540,395.504,179.233,24.461,153.603
C02581=1096.492,446.294,395.548,179.233,24.448,153.600
C02582=1096.486,446.048,395.592,179.232,24.436,153.597
C02583=1096.480,445.802,395.635,179.230,24.422,153.594
C02584=1096.473,445.556,395.679,179.229,24.409,153.591
C02585=1096.467,445.310,395.723,179.228,24.396,153.587
C02586=1096.460,445.064,395.767,179.226,24.383,153.584
C02587=1096.454,444.818,395.811,179.224,24.370,153.581
C02588=1096.448,444.571,395.854,179.223,24.357,153.578
C02589=1096.442,444.326,395.897,179.220,24.344,153.575
C02590=1096.436,444.080,395.941,179.218,24.331,153.572
C02591=1096.429,443.834,395.985,179.216,24.318,153.569
C02592=1096.423,443.588,396.029,179.213,24.304,153.566
C02593=1096.417,443.341,396.072,179.210,24.291,153.563
C02594=1096.410,443.095,396.116,179.209,24.279,153.560
C02595=1096.404,442.850,396.159,179.206,24.265,153.557
C02596=1096.397,442.604,396.202,179.203,24.253,153.554
C02597=1096.391,442.358,396.246,179.201,24.240,153.551
C02598=1096.385,442.111,396.289,179.198,24.227,153.548
C02599=1096.379,441.865,396.333,179.196,24.214,153.545
C02600=1096.373,441.620,396.376,179.193,24.201,153.543
C02601=1096.366,441.374,396.419,179.191,24.189,153.540
C02602=1096.359,441.128,396.463,179.188,24.176,153.537
C02603=1096.354,440.882,396.505,179.185,24.163,153.534
C02604=1096.348,440.635,396.549,179.183,24.151,153.531
C02605=1096.341,440.390,396.592,179.180,24.138,153.528
C02606=1096.334,440.143,396.635,179.178,24.126,153.526
C02607=1096.329,439.898,396.678,179.176,24.114,153.523
C02608=1096.322,439.652,396.721,179.173,24.101,153.520
C02609=1096.316,439.405,396.764,179.170,24.089,153.517
C02610=1096.310,439.158,396.807,179.167,24.076,153.515
C02611=1096.303,438.913,396.850,179.165,24.064,153.512
C02612=1096.297,438.667,396.893,179.162,24.052,153.509
C02613=1096.290,438.420,396.936,179.159,24.040,153.507
C02614=1096.283,438.156,396.982,179.157,24.027,153.504
C02615=1096.277,437.893,397.028,179.154,24.014,153.501
C02616=1096.271,437.629,397.074,179.151,24.002,153.498
C02617=1096.263,437.364,397.120,179.149,23.989,153.495
C02618=1096.257,437.118,397.163,179.146,23.977,153.492
C02619=1096.251,436.872,397.205,179.144,23.965,153.490
C02620=1096.245,436.626,397.248,179.141,23.953,153.487
C02621=1096.238,436.379,397.291,179.138,23.941,153.484
C02622=1096.232,436.133,397.333,179.136,23.930,153.482
C02623=1096.226,435.887,397.376,179.133,23.918,153.479
C02624=1096.220,435.641,397.419,179.131,23.906,153.477
C02625=1096.213,435.395,397.461,179.128,23.894,153.474
C02626=1096.208,435.149,397.503,179.126,23.883,153.471
C02627=1096.201,434.902,397.546,179.123,23.872,153.469
C02628=1096.196,434.656,397.589,179.121,23.860,153.466
C02629=1096.189,434.410,397.631,179.118,23.849,153.464
C02630=1096.183,434.164,397.674,179.115,23.837,153.461
C02631=1096.177,433.917,397.716,179.112,23.826,153.459
C02632=1096.170,433.672,397.758,179.109,23.814,153.456
C02633=1096.164,433.425,397.801,179.107,23.803,153.454
C02634=1096.158,433.179,397.842,179.104,23.792,153.452
C02635=1096.152,432.932,397.886,179.102,23.781,153.449
C02636=1096.146,432.686,397.927,179.100,23.769,153.447
C02637=1096.140,432.440,397.970,179.097,23.758,153.444
C02638=1096.133,432.194,398.012,179.094,23.747,153.442
C02639=1096.127,431.947,398.054,179.091,23.736,153.439
C02640=1096.121,431.701,398.096,179.089,23.725,153.437
C02641=1096.115,431.455,398.138,179.086,23.714,153.435
C02642=1096.109,431.208,398.180,179.084,23.703,153.432
C02643=1096.102,430.963,398.222,179.081,23.693,153.430
C02644=1096.097,430.715,398.264,179.078,23.681,153.427
C02645=1096.090,430.470,398.306,179.076,23.671,153.425
C02646=1096.084,430.224,398.348,179.073,23.660,153.423
C02647=1096.078,429.977,398.390,179.070,23.649,153.420
C02648=1096.072,429.731,398.432,179.068,23.638,153.418
C02649=1096.065,429.484,398.474,179.065,23.628,153.416
C02650=1096.060,429.238,398.516,179.062,23.617,153.414
C02651=1096.054,428.992,398.557,179.060,23.607,153.411
C02652=1096.047,428.745,398.599,179.057,23.596,153.409
C02653=1096.041,428.499,398.641,179.054,23.586,153.407
C02654=1096.035,428.253,398.683,179.052,23.575,153.405
C02655=1096.029,428.006,398.724,179.049,23.564,153.402
C02656=1096.023,427.760,398.766,179.046,23.554,153.400
C02657=1096.017,427.514,398.807,179.044,23.544,153.398
C02658=1096.010,427.267,398.849,179.041,23.533,153.396
C02659=1096.004,427.020,398.891,179.038,23.524,153.394
C02660=1095.998,426.774,398.932,179.036,23.513,153.391
C02661=1095.992,426.527,398.974,179.033,23.503,153.389
C02662=1095.985,426.281,399.015,179.030,23.492,153.387
C02663=1095.979,426.035,399.056,179.027,23.483,153.385
C02664=1095.973,425.789,399.098,179.025,23.472,153.383
C02665=1095.967,425.542,399.140,179.022,23.463,153.381
C02666=1095.962,425.316,399.177,179.020,23.453,153.379
C02667=1095.956,425.089,399.215,179.017,23.444,153.377
C02668=1095.950,424.862,399.253,179.015,23.435,153.375
C02669=1095.945,424.634,399.292,179.012,23.426,153.373
C02670=1095.939,424.408,399.330,179.010,23.416,153.371
C02671=1095.933,424.182,399.368,179.008,23.407,153.369
C02672=1095.928,423.955,399.405,179.005,23.398,153.367
C02673=1095.922,423.728,399.444,179.002,23.389,153.365
C02674=1095.916,423.482,399.485,179.000,23.379,153.363
C02675=1095.910,423.236,399.525,178.997,23.370,153.361
C02676=1095.904,422.989,399.567,178.995,23.360,153.359
C02677=1095.898,422.742,399.608,178.992,23.350,153.357
C02678=1095.892,422.496,399.649,178.990,23.341,153.355
C02679=1095.885,422.250,399.690,178.986,23.330,153.353
C02680=1095.880,422.003,399.731,178.983,23.321,153.351
C02681=1095.873,421.756,399.773,178.981,23.312,153.349
C02682=1095.867,421.510,399.813,178.978,23.302,153.347
C02683=1095.861,421.263,399.854,178.976,23.292,153.345
C02684=1095.855,421.016,399.895,178.973,23.283,153.343
C02685=1095.849,420.770,399.935,178.970,23.274,153.341
C02686=1095.843,420.524,399.977,178.968,23.264,153.339
C02687=1095.837,420.277,400.017,178.965,23.255,153.337
C02688=1095.830,420.031,400.058,178.962,23.245,153.335
C02689=1095.824,419.784,400.099,178.960,23.236,153.333
C02690=1095.818,419.537,400.140,178.957,23.227,153.331
C02691=1095.812,419.290,400.180,178.954,23.218,153.329
C02692=1095.806,419.044,400.222,178.951,23.209,153.327
C02693=1095.800,418.797,400.262,178.949,23.199,153.325
C02694=1095.794,418.551,400.303,178.946,23.190,153.324
C02695=1095.788,418.304,400.343,178.943,23.181,153.322
C02696=1095.782,418.058,400.384,178.940,23.172,153.320
C02697=1095.776,417.811,400.424,178.938,23.163,153.318
C02698=1095.770,417.565,400.465,178.935,23.154,153.316
C02699=1095.764,417.318,400.506,178.932,23.145,153.314
C02700=1095.758,417.071,400.546,178.929,23.136,153.312
C02701=1095.752,416.824,400.587,178.927,23.126,153.311
C02702=1095.746,416.578,400.627,178.924,23.117,153.309
C02703=1095.740,416.331,400.668,178.921,23.108,153.307
C02704=1095.734,416.085,400.708,178.918,23.100,153.305
C02705=1095.727,415.838,400.748,178.916,23.091,153.303
C02706=1095.722,415.591,400.789,178.914,23.082,153.302
C02707=1095.715,415.345,400.829,178.911,23.074,153.300
C02708=1095.709,415.098,400.869,178.908,23.065,153.298
C02709=1095.703,414.852,400.909,178.905,23.056,153.296
C02710=1095.697,414.605,400.950,178.902,23.047,153.295
C02711=1095.691,414.358,400.989,178.899,23.039,153.293
C02712=1095.685,414.111,401.029,178.897,23.030,153.291
C02713=1095.679,413.864,401.070,178.894,23.022,153.289
C02714=1095.673,413.618,401.110,178.892,23.013,153.288
C02715=1095.666,413.371,401.150,178.889,23.005,153.286
C02716=1095.661,413.125,401.190,178.886,22.996,153.284
C02717=1095.655,412.878,401.230,178.884,22.988,153.283
C02718=1095.649,412.632,401.270,178.881,22.979,153.281
C02719=1095.643,412.384,401.310,178.878,22.971,153.279
C02720=1095.636,412.138,401.350,178.875,22.962,153.277
C02721=1095.630,411.891,401.390,178.872,22.954,153.276
C02722=1095.625,411.672,401.426,178.870,22.946,153.274
C02723=1095.619,411.452,401.461,178.867,22.939,153.273
C02724=1095.615,411.232,401.496,178.865,22.932,153.271
C02725=1095.608,411.013,401.532,178.863,22.924,153.270
C02726=1095.604,410.794,401.568,178.860,22.917,153.268
C02727=1095.598,410.574,401.603,178.858,22.909,153.267
C02728=1095.593,410.354,401.638,178.856,22.902,153.266
C02729=1095.587,410.134,401.673,178.853,22.895,153.264
C02730=1095.582,409.887,401.714,178.850,22.886,153.262
C02731=1095.576,409.640,401.754,178.847,22.878,153.261
C02732=1095.570,409.394,401.793,178.845,22.870,153.259
C02733=1095.564,409.147,401.833,178.842,22.862,153.258
C02734=1095.558,408.900,401.872,178.839,22.854,153.256
C02735=1095.551,408.654,401.912,178.837,22.846,153.254
C02736=1095.546,408.407,401.951,178.834,22.838,153.253
C02737=1095.540,408.160,401.991,178.831,22.830,153.251
C02738=1095.533,407.914,402.031,178.829,22.822,153.250
C02739=1095.528,407.667,402.070,178.826,22.814,153.248
C02740=1095.522,407.420,402.110,178.823,22.806,153.247
C02741=1095.516,407.173,402.149,178.820,22.798,153.245
C02742=1095.509,406.926,402.189,178.817,22.790,153.243
C02743=1095.504,406.680,402.228,178.815,22.783,153.242
C02744=1095.498,406.433,402.268,178.812,22.774,153.240
C02745=1095.492,406.186,402.307,178.809,22.766,153.239
C02746=1095.486,405.939,402.346,178.807,22.759,153.237
C02747=1095.480,405.692,402.386,178.804,22.751,153.236
C02748=1095.474,405.445,402.425,178.801,22.744,153.234
C02749=1095.468,405.199,402.465,178.798,22.735,153.233
C02750=1095.462,404.952,402.504,178.796,22.728,153.231
C02751=1095.456,404.705,402.544,178.793,22.720,153.230
C02752=1095.451,404.458,402.583,178.791,22.713,153.228
C02753=1095.444,404.212,402.621,178.787,22.705,153.227
C02754=1095.438,403.964,402.661,178.785,22.698,153.226
C02755=1095.433,403.717,402.699,178.782,22.690,153.224
C02756=1095.427,403.470,402.739,178.779,22.683,153.223
C02757=1095.420,403.223,402.778,178.776,22.675,153.221
C02758=1095.414,402.977,402.817,178.774,22.668,153.220
C02759=1095.408,402.730,402.856,178.771,22.660,153.218
C02760=1095.403,402.483,402.895,178.768,22.653,153.217
C02761=1095.396,402.237,402.934,178.765,22.645,153.216
C02762=1095.390,401.989,402.973,178.763,22.638,153.214
C02763=1095.385,401.742,403.012,178.760,22.630,153.213
C02764=1095.378,401.496,403.051,178.757,22.623,153.211
C02765=1095.373,401.249,403.090,178.754,22.616,153.210
C02766=1095.366,401.002,403.129,178.752,22.608,153.209
C02767=1095.361,400.755,403.167,178.749,22.601,153.207
C02768=1095.354,400.508,403.206,178.746,22.594,153.206
C02769=1095.349,400.262,403.245,178.744,22.587,153.205
C02770=1095.343,400.014,403.284,178.740,22.579,153.203
C02771=1095.337,399.768,403.323,178.738,22.572,153.202
C02772=1095.331,399.520,403.361,178.736,22.565,153.200
C02773=1095.325,399.274,403.400,178.732,22.558,153.199
C02774=1095.319,399.027,403.439,178.730,22.551,153.198
C02775=1095.313,398.780,403.477,178.726,22.544,153.197
C02776=1095.307,398.533,403.516,178.724,22.537,153.195
C02777=1095.301,398.286,403.554,178.722,22.530,153.194
C02778=1095.296,398.067,403.589,178.719,22.523,153.193
C02779=1095.291,397.847,403.623,178.716,22.517,153.192
C02780=1095.285,397.628,403.658,178.713,22.511,153.190
C02781=1095.280,397.408,403.691,178.712,22.505,153.189
C02782=1095.274,397.189,403.726,178.709,22.498,153.188
C02783=1095.270,396.970,403.760,178.706,22.492,153.187
C02784=1095.264,396.751,403.794,178.705,22.486,153.186
C02785=1095.259,396.531,403.828,178.702,22.480,153.185
C02786=1095.254,396.284,403.867,178.699,22.473,153.183
C02787=1095.247,396.037,403.906,178.696,22.466,153.182
C02788=1095.241,395.791,403.943,178.693,22.459,153.181
C02789=1095.236,395.543,403.982,178.691,22.453,153.180
C02790=1095.229,395.297,404.020,178.687,22.445,153.178
C02791=1095.224,395.050,404.059,178.685,22.439,153.177
C02792=1095.218,394.803,404.097,178.682,22.432,153.176
C02793=1095.211,394.555,404.135,178.679,22.425,153.175
C02794=1095.206,394.309,404.174,178.676,22.418,153.173
C02795=1095.199,394.062,404.212,178.674,22.412,153.172
C02796=1095.193,393.815,404.250,178.671,22.405,153.171
C02797=1095.188,393.568,404.287,178.668,22.398,153.170
C02798=1095.182,393.321,404.326,178.665,22.392,153.169
C02799=1095.176,393.074,404.364,178.663,22.385,153.168
C02800=1095.170,392.827,404.402,178.660,22.379,153.166
C02801=1095.165,392.580,404.441,178.657,22.372,153.165
C02802=1095.158,392.333,404.479,178.654,22.365,153.164
C02803=1095.152,392.086,404.517,178.651,22.359,153.163
C02804=1095.146,391.839,404.554,178.649,22.352,153.162
C02805=1095.140,391.593,404.592,178.646,22.346,153.160
C02806=1095.134,391.345,404.630,178.643,22.339,153.159
C02807=1095.128,391.099,404.668,178.640,22.333,153.158
C02808=1095.122,390.852,404.706,178.637,22.327,153.157
C02809=1095.117,390.605,404.744,178.635,22.320,153.156
C02810=1095.110,390.357,404.782,178.632,22.314,153.155
C02811=1095.104,390.111,404.820,178.628,22.307,153.154
C02812=1095.099,389.863,404.857,178.626,22.301,153.153
C02813=1095.093,389.616,404.895,178.623,22.295,153.151
C02814=1095.086,389.369,404.933,178.620,22.289,153.150
C02815=1095.081,389.122,404.971,178.618,22.282,153.149
C02816=1095.075,388.875,405.008,178.614,22.276,153.148
C02817=1095.069,388.629,405.046,178.611,22.269,153.147
C02818=1095.063,388.381,405.083,178.609,22.263,153.146
C02819=1095.057,388.135,405.121,178.606,22.257,153.145
C02820=1095.051,387.887,405.159,178.603,22.251,153.144
C02821=1095.045,387.640,405.197,178.601,22.244,153.143
C02822=1095.039,387.393,405.234,178.597,22.238,153.142
C02823=1095.033,387.146,405.272,178.594,22.232,153.141
C02824=1095.027,386.900,405.309,178.591,22.226,153.140
C02825=1095.021,386.653,405.347,178.589,22.220,153.138
C02826=1095.016,386.406,405.384,178.586,22.214,153.137
C02827=1095.010,386.159,405.422,178.583,22.208,153.136
C02828=1095.004,385.911,405.459,178.580,22.202,153.135
C02829=1094.998,385.665,405.496,178.577,22.195,153.134
C02830=1094.992,385.418,405.533,178.574,22.189,153.133
C02831=1094.986,385.171,405.571,178.571,22.183,153.132
C02832=1094.980,384.923,405.609,178.569,22.177,153.131
C02833=1094.975,384.677,405.646,178.566,22.171,153.130
C02834=1094.970,384.463,405.678,178.564,22.166,153.129
C02835=1094.964,384.251,405.710,178.560,22.160,153.128
C02836=1094.959,384.037,405.743,178.558,22.155,153.127
C02837=1094.955,383.825,405.775,178.555,22.150,153.127
C02838=1094.949,383.612,405.807,178.553,22.145,153.126
C02839=1094.944,383.399,405.839,178.551,22.140,153.125
C02840=1094.939,383.186,405.872,178.548,22.135,153.124
C02841=1094.934,382.974,405.903,178.546,22.130,153.123
C02842=1094.929,382.726,405.940,178.543,22.123,153.122
C02843=1094.923,382.479,405.977,178.540,22.118,153.121
C02844=1094.917,382.232,406.014,178.537,22.112,153.120
C02845=1094.911,381.985,406.052,178.535,22.106,153.119
C02846=1094.905,381.738,406.089,178.532,22.100,153.118
C02847=1094.899,381.491,406.125,178.529,22.094,153.117
C02848=1094.893,381.244,406.163,178.526,22.089,153.116
C02849=1094.887,380.997,406.200,178.523,22.083,153.115
C02850=1094.881,380.749,406.236,178.520,22.077,153.114
C02851=1094.875,380.502,406.273,178.517,22.072,153.113
C02852=1094.870,380.255,406.310,178.514,22.066,153.113
C02853=1094.863,380.008,406.347,178.512,22.060,153.112
C02854=1094.858,379.761,406.385,178.509,22.054,153.111
C02855=1094.851,379.514,406.421,178.506,22.049,153.110
C02856=1094.846,379.267,406.458,178.503,22.043,153.109
C02857=1094.840,379.019,406.495,178.500,22.037,153.108
C02858=1094.834,378.772,406.531,178.497,22.032,153.107
C02859=1094.828,378.525,406.569,178.494,22.026,153.106
C02860=1094.822,378.278,406.605,178.491,22.021,153.105
C02861=1094.817,378.031,406.642,178.488,22.015,153.104
C02862=1094.811,377.784,406.679,178.485,22.009,153.103
C02863=1094.805,377.537,406.715,178.482,22.004,153.103
C02864=1094.799,377.289,406.752,178.479,21.998,153.102
C02865=1094.793,377.042,406.789,178.476,21.993,153.101
C02866=1094.787,376.795,406.826,178.473,21.987,153.100
C02867=1094.781,376.548,406.862,178.471,21.981,153.099
C02868=1094.776,376.301,406.899,178.468,21.976,153.098
C02869=1094.770,376.054,406.935,178.465,21.970,153.097
C02870=1094.764,375.806,406.972,178.462,21.965,153.096
C02871=1094.758,375.559,407.008,178.459,21.959,153.095
C02872=1094.752,375.312,407.045,178.456,21.954,153.095
C02873=1094.747,375.065,407.081,178.453,21.948,153.094
C02874=1094.741,374.818,407.118,178.450,21.943,153.093
C02875=1094.735,374.570,407.154,178.447,21.937,153.092
C02876=1094.729,374.323,407.191,178.444,21.932,153.091
C02877=1094.723,374.076,407.227,178.441,21.927,153.090
C02878=1094.717,373.829,407.264,178.439,21.921,153.089
C02879=1094.712,373.581,407.300,178.436,21.916,153.089
C02880=1094.706,373.334,407.336,178.432,21.911,153.088
C02881=1094.699,373.087,407.373,178.430,21.906,153.087
C02882=1094.694,372.839,407.409,178.426,21.900,153.086
C02883=1094.688,372.592,407.445,178.423,21.895,153.085
C02884=1094.682,372.345,407.481,178.420,21.890,153.085
C02885=1094.676,372.098,407.517,178.417,21.884,153.084
C02886=1094.670,371.851,407.554,178.414,21.879,153.083
C02887=1094.664,371.603,407.590,178.412,21.874,153.082
C02888=1094.659,371.357,407.626,178.409,21.869,153.081
C02889=1094.653,371.109,407.662,178.406,21.864,153.081
C02890=1094.643,370.711,407.721,178.401,21.856,153.079
C02891=1094.634,370.312,407.778,178.396,21.847,153.078
C02892=1094.624,369.914,407.837,178.391,21.839,153.077
C02893=1094.615,369.516,407.895,178.387,21.831,153.076
C02894=1094.609,369.268,407.930,178.384,21.826,153.075
C02895=1094.604,369.021,407.967,178.381,21.820,153.074
C02896=1094.598,368.773,408.003,178.378,21.815,153.073
C02897=1094.592,368.526,408.038,178.375,21.810,153.073
C02898=1094.586,368.279,408.075,178.371,21.805,153.072
C02899=1094.580,368.032,408.110,178.369,21.800,153.071
C02900=1094.574,367.784,408.146,178.366,21.795,153.070
C02901=1094.568,367.537,408.182,178.363,21.790,153.070
C02902=1094.563,367.290,408.218,178.360,21.785,153.069
C02903=1094.557,367.042,408.254,178.357,21.780,153.068
C02904=1094.551,366.795,408.290,178.355,21.775,153.067
C02905=1094.546,366.548,408.325,178.351,21.770,153.067
C02906=1094.540,366.300,408.361,178.348,21.765,153.066
C02907=1094.534,366.054,408.397,178.345,21.760,153.065
C02908=1094.528,365.806,408.433,178.342,21.755,153.064
C02909=1094.522,365.558,408.468,178.340,21.750,153.064
C02910=1094.517,365.311,408.504,178.336,21.745,153.063
C02911=1094.510,365.064,408.540,178.333,21.740,153.062
C02912=1094.504,364.816,408.575,178.330,21.735,153.062
C02913=1094.499,364.569,408.611,178.327,21.730,153.061
C02914=1094.493,364.321,408.646,178.325,21.726,153.060
C02915=1094.488,364.074,408.682,178.321,21.721,153.060
C02916=1094.482,363.827,408.717,178.318,21.716,153.059
C02917=1094.476,363.580,408.753,178.315,21.711,153.058
C02918=1094.470,363.332,408.789,178.313,21.707,153.058
C02919=1094.464,363.084,408.824,178.309,21.702,153.057
C02920=1094.459,362.837,408.860,178.306,21.697,153.056
C02921=1094.452,362.590,408.895,178.303,21.692,153.056
C02922=1094.446,362.343,408.930,178.301,21.687,153.055
C02923=1094.441,362.095,408.965,178.297,21.683,153.054
C02924=1094.435,361.848,409.001,178.294,21.678,153.054
C02925=1094.429,361.600,409.036,178.291,21.673,153.053
C02926=1094.424,361.353,409.072,178.289,21.669,153.052
C02927=1094.418,361.105,409.107,178.285,21.664,153.052
C02928=1094.412,360.859,409.142,178.282,21.659,153.051
C02929=1094.406,360.610,409.177,178.280,21.654,153.050
C02930=1094.400,360.363,409.212,178.276,21.650,153.050
C02931=1094.394,360.116,409.248,178.273,21.645,153.049
C02932=1094.389,359.868,409.283,178.270,21.640,153.048
C02933=1094.383,359.621,409.318,178.267,21.636,153.048
C02934=1094.377,359.374,409.353,178.264,21.631,153.047
C02935=1094.371,359.126,409.389,178.261,21.626,153.047
C02936=1094.365,358.879,409.423,178.258,21.622,153.046
C02937=1094.359,358.631,409.459,178.255,21.618,153.045
C02938=1094.354,358.384,409.494,178.252,21.613,153.045
C02939=1094.347,358.136,409.529,178.249,21.609,153.044
C02940=1094.342,357.889,409.564,178.246,21.604,153.044
C02941=1094.336,357.641,409.599,178.243,21.599,153.043
C02942=1094.327,357.258,409.653,178.239,21.592,153.042
C02943=1094.318,356.874,409.707,178.234,21.585,153.041
C02944=1094.309,356.491,409.761,178.229,21.578,153.040
C02945=1094.300,356.108,409.815,178.224,21.571,153.039
C02946=1094.295,355.861,409.851,178.222,21.567,153.039
C02947=1094.289,355.614,409.885,178.218,21.562,153.038
C02948=1094.283,355.365,409.920,178.215,21.557,153.037
C02949=1094.277,355.119,409.955,178.213,21.554,153.037
C02950=1094.271,354.871,409.990,178.209,21.549,153.036
C02951=1094.266,354.623,410.024,178.206,21.544,153.036
C02952=1094.260,354.376,410.059,178.203,21.540,153.035
C02953=1094.254,354.128,410.094,178.200,21.536,153.035
C02954=1094.248,353.881,410.128,178.197,21.531,153.034
C02955=1094.243,353.634,410.163,178.194,21.527,153.033
C02956=1094.236,353.386,410.198,178.191,21.522,153.033
C02957=1094.231,353.138,410.232,178.188,21.518,153.032
C02958=1094.225,352.891,410.267,178.185,21.514,153.032
C02959=1094.219,352.643,410.302,178.182,21.509,153.031
C02960=1094.214,352.396,410.336,178.179,21.505,153.031
C02961=1094.208,352.149,410.370,178.176,21.501,153.030
C02962=1094.202,351.900,410.405,178.172,21.496,153.030
C02963=1094.196,351.653,410.439,178.170,21.492,153.029
C02964=1094.191,351.405,410.474,178.166,21.488,153.029
C02965=1094.184,351.157,410.509,178.164,21.484,153.028
C02966=1094.178,350.911,410.543,178.160,21.479,153.028
C02967=1094.173,350.663,410.578,178.157,21.475,153.027
C02968=1094.167,350.415,410.612,178.155,21.471,153.026
C02969=1094.161,350.168,410.646,178.151,21.467,153.026
C02970=1094.156,349.920,410.681,178.148,21.463,153.026
C02971=1094.150,349.673,410.715,178.145,21.458,153.025
C02972=1094.144,349.425,410.750,178.143,21.454,153.024
C02973=1094.138,349.177,410.784,178.139,21.450,153.024
C02974=1094.132,348.930,410.818,178.136,21.446,153.023
C02975=1094.127,348.683,410.852,178.133,21.441,153.023
C02976=1094.121,348.435,410.887,178.130,21.437,153.022
C02977=1094.115,348.187,410.921,178.127,21.433,153.022
C02978=1094.109,347.939,410.955,178.124,21.429,153.021
C02979=1094.104,347.692,410.989,178.121,21.425,153.021
C02980=1094.098,347.445,411.023,178.118,21.421,153.020
C02981=1094.092,347.197,411.058,178.115,21.417,153.020
C02982=1094.086,346.949,411.092,178.112,21.412,153.019
C02983=1094.081,346.702,411.126,178.108,21.408,153.019
C02984=1094.075,346.454,411.160,178.106,21.404,153.018
C02985=1094.070,346.206,411.194,178.102,21.400,153.018
C02986=1094.063,345.959,411.228,178.100,21.396,153.017
C02987=1094.057,345.711,411.262,178.096,21.392,153.017
C02988=1094.052,345.463,411.296,178.094,21.388,153.017
C02989=1094.047,345.216,411.330,178.090,21.383,153.016
C02990=1094.041,344.968,411.364,178.088,21.380,153.016
C02991=1094.035,344.721,411.398,178.084,21.375,153.015
C02992=1094.029,344.473,411.432,178.081,21.372,153.015
C02993=1094.023,344.225,411.466,178.078,21.368,153.014
C02994=1094.015,343.845,411.518,178.073,21.361,153.014
C02995=1094.005,343.464,411.570,178.068,21.355,153.013
C02996=1093.997,343.083,411.622,178.064,21.349,153.012
C02997=1093.987,342.703,411.674,178.059,21.344,153.012
C02998=1093.982,342.454,411.709,178.056,21.339,153.011
C02999=1093.976,342.207,411.742,178.053,21.336,153.011
C03000=1093.970,341.959,411.776,178.050,21.331,153.010
C03001=1093.965,341.711,411.809,178.047,21.328,153.010
C03002=1093.959,341.464,411.844,178.044,21.324,153.009
C03003=1093.953,341.216,411.876,178.041,21.320,153.009
C03004=1093.947,340.969,411.910,178.037,21.316,153.009
C03005=1093.941,340.721,411.944,178.035,21.312,153.008
C03006=1093.936,340.473,411.977,178.031,21.308,153.008
C03007=1093.930,340.226,412.011,178.029,21.304,153.007
C03008=1093.924,339.978,412.044,178.025,21.300,153.007
C03009=1093.919,339.730,412.078,178.022,21.297,153.006
C03010=1093.913,339.483,412.112,178.019,21.292,153.006
C03011=1093.907,339.235,412.145,178.016,21.288,153.005
C03012=1093.902,338.987,412.178,178.014,21.285,153.005
C03013=1093.896,338.740,412.213,178.010,21.281,153.005
C03014=1093.890,338.492,412.246,178.007,21.277,153.004
C03015=1093.885,338.244,412.279,178.004,21.273,153.004
C03016=1093.879,337.996,412.313,178.001,21.270,153.004
C03017=1093.872,337.749,412.346,177.997,21.266,153.003
C03018=1093.866,337.501,412.380,177.995,21.262,153.003
C03019=1093.861,337.253,412.413,177.992,21.259,153.002
C03020=1093.855,337.005,412.446,177.988,21.255,153.002
C03021=1093.849,336.757,412.479,177.986,21.251,153.002
C03022=1093.843,336.510,412.513,177.982,21.247,153.001
C03023=1093.838,336.263,412.546,177.979,21.244,153.001
C03024=1093.833,336.015,412.579,177.976,21.239,153.000
C03025=1093.826,335.767,412.612,177.973,21.236,153.000
C03026=1093.821,335.519,412.646,177.970,21.233,153.000
C03027=1093.815,335.271,412.679,177.967,21.228,152.999
C03028=1093.810,335.024,412.712,177.964,21.225,152.999
C03029=1093.803,334.776,412.745,177.960,21.221,152.999
C03030=1093.798,334.528,412.778,177.958,21.218,152.998
C03031=1093.792,334.280,412.812,177.955,21.214,152.998
C03032=1093.786,334.033,412.844,177.951,21.210,152.997
C03033=1093.780,333.785,412.878,177.949,21.207,152.997
C03034=1093.775,333.537,412.911,177.946,21.203,152.997
C03035=1093.769,333.289,412.944,177.942,21.199,152.996
C03036=1093.763,333.041,412.977,177.940,21.195,152.996
C03037=1093.758,332.794,413.010,177.936,21.192,152.996
C03038=1093.752,332.546,413.043,177.933,21.188,152.995
C03039=1093.746,332.299,413.076,177.930,21.185,152.995
C03040=1093.741,332.050,413.109,177.927,21.181,152.995
C03041=1093.735,331.802,413.142,177.924,21.178,152.994
C03042=1093.729,331.554,413.175,177.921,21.174,152.994
C03043=1093.723,331.307,413.208,177.917,21.170,152.994
C03044=1093.717,331.059,413.240,177.915,21.167,152.993
C03045=1093.711,330.811,413.274,177.912,21.164,152.993
C03046=1093.703,330.424,413.324,177.907,21.158,152.993
C03047=1093.692,330.038,413.375,177.902,21.152,152.992
C03048=1093.684,329.651,413.427,177.897,21.147,152.992
C03049=1093.675,329.265,413.477,177.893,21.142,152.991
C03050=1093.669,329.017,413.510,177.889,21.138,152.991
C03051=1093.663,328.769,413.543,177.886,21.135,152.990
C03052=1093.657,328.521,413.575,177.883,21.131,152.990
C03053=1093.651,328.273,413.608,177.880,21.128,152.990
C03054=1093.646,328.025,413.641,177.877,21.124,152.989
C03055=1093.640,327.778,413.673,177.874,21.121,152.989
C03056=1093.634,327.530,413.706,177.870,21.117,152.989
C03057=1093.629,327.282,413.738,177.867,21.114,152.989
C03058=1093.622,327.034,413.771,177.865,21.111,152.988
C03059=1093.616,326.787,413.804,177.861,21.107,152.988
C03060=1093.611,326.539,413.836,177.858,21.104,152.988
C03061=1093.605,326.291,413.869,177.855,21.100,152.987
C03062=1093.599,326.043,413.901,177.852,21.097,152.987
C03063=1093.594,325.795,413.934,177.849,21.093,152.987
C03064=1093.588,325.548,413.966,177.846,21.090,152.987
C03065=1093.582,325.299,413.998,177.843,21.087,152.986
C03066=1093.576,325.052,414.031,177.839,21.083,152.986
C03067=1093.571,324.803,414.063,177.836,21.080,152.986
C03068=1093.565,324.556,414.096,177.834,21.077,152.985
C03069=1093.559,324.308,414.128,177.831,21.073,152.985
C03070=1093.553,324.060,414.160,177.827,21.070,152.985
C03071=1093.548,323.813,414.193,177.824,21.066,152.985
C03072=1093.542,323.564,414.225,177.821,21.063,152.984
C03073=1093.536,323.316,414.257,177.818,21.060,152.984
C03074=1093.530,323.069,414.289,177.815,21.056,152.984
C03075=1093.525,322.821,414.322,177.812,21.053,152.983
C03076=1093.519,322.573,414.354,177.809,21.050,152.983
C03077=1093.513,322.326,414.386,177.806,21.046,152.983
C03078=1093.507,322.077,414.418,177.802,21.043,152.983
C03079=1093.501,321.829,414.450,177.800,21.040,152.982
C03080=1093.497,321.581,414.483,177.797,21.037,152.982
C03081=1093.490,321.334,414.515,177.794,21.033,152.982
C03082=1093.485,321.086,414.547,177.790,21.029,152.981
C03083=1093.479,320.838,414.579,177.787,21.026,152.981
C03084=1093.473,320.590,414.611,177.784,21.023,152.981
C03085=1093.468,320.342,414.643,177.781,21.020,152.981
C03086=1093.462,320.094,414.675,177.778,21.016,152.980
C03087=1093.457,319.846,414.707,177.775,21.013,152.980
C03088=1093.451,319.599,414.740,177.772,21.010,152.980
C03089=1093.445,319.351,414.771,177.769,21.007,152.980
C03090=1093.439,319.103,414.803,177.765,21.003,152.979
C03091=1093.434,318.856,414.835,177.762,21.000,152.979
C03092=1093.429,318.607,414.868,177.760,20.997,152.979
C03093=1093.423,318.359,414.900,177.757,20.994,152.979
C03094=1093.417,318.111,414.931,177.754,20.990,152.978
C03095=1093.411,317.863,414.963,177.750,20.987,152.978
C03096=1093.406,317.616,414.995,177.747,20.984,152.978
C03097=1093.401,317.368,415.027,177.744,20.981,152.978
C03098=1093.391,316.974,415.078,177.739,20.975,152.977
C03099=1093.383,316.580,415.129,177.735,20.970,152.977
C03100=1093.373,316.186,415.178,177.730,20.965,152.976
C03101=1093.365,315.793,415.229,177.725,20.960,152.976
C03102=1093.359,315.545,415.260,177.722,20.957,152.976
C03103=1093.354,315.298,415.292,177.719,20.954,152.975
C03104=1093.348,315.049,415.324,177.716,20.950,152.975
C03105=1093.343,314.801,415.355,177.712,20.947,152.975
C03106=1093.337,314.553,415.387,177.709,20.944,152.975
C03107=1093.330,314.305,415.418,177.706,20.941,152.975
C03108=1093.325,314.058,415.450,177.703,20.938,152.974
C03109=1093.319,313.809,415.482,177.700,20.935,152.974
C03110=1093.313,313.562,415.512,177.697,20.932,152.974
C03111=1093.307,313.313,415.544,177.693,20.929,152.974
C03112=1093.302,313.066,415.576,177.690,20.926,152.974
C03113=1093.296,312.817,415.607,177.687,20.923,152.973
C03114=1093.290,312.570,415.639,177.684,20.920,152.973
C03115=1093.284,312.322,415.670,177.681,20.917,152.973
C03116=1093.278,312.074,415.702,177.678,20.914,152.973
C03117=1093.273,311.826,415.733,177.675,20.911,152.973
C03118=1093.267,311.578,415.765,177.672,20.908,152.973
C03119=1093.262,311.330,415.796,177.669,20.905,152.972
C03120=1093.255,311.082,415.827,177.666,20.902,152.972
C03121=1093.249,310.834,415.859,177.663,20.899,152.972
C03122=1093.244,310.587,415.889,177.660,20.896,152.972
C03123=1093.238,310.338,415.921,177.657,20.893,152.972
C03124=1093.233,310.090,415.952,177.653,20.889,152.971
C03125=1093.226,309.842,415.983,177.650,20.886,152.971
C03126=1093.221,309.594,416.014,177.647,20.883,152.971
C03127=1093.215,309.347,416.045,177.644,20.881,152.971
C03128=1093.209,309.098,416.077,177.641,20.878,152.971
C03129=1093.204,308.851,416.108,177.638,20.875,152.970
C03130=1093.198,308.603,416.139,177.635,20.872,152.970
C03131=1093.192,308.355,416.171,177.631,20.868,152.970
C03132=1093.186,308.107,416.201,177.628,20.865,152.970
C03133=1093.181,307.859,416.233,177.625,20.862,152.970
C03134=1093.174,307.611,416.263,177.622,20.859,152.969
C03135=1093.169,307.363,416.294,177.619,20.856,152.969
C03136=1093.164,307.115,416.326,177.616,20.853,152.969
C03137=1093.158,306.867,416.356,177.613,20.851,152.969
C03138=1093.152,306.619,416.388,177.610,20.848,152.969
C03139=1093.146,306.371,416.419,177.606,20.845,152.969
C03140=1093.141,306.123,416.450,177.603,20.842,152.968
C03141=1093.135,305.875,416.480,177.600,20.839,152.968
C03142=1093.129,305.627,416.512,177.597,20.836,152.968
C03143=1093.123,305.379,416.542,177.594,20.833,152.968
C03144=1093.118,305.131,416.573,177.591,20.830,152.968
C03145=1093.112,304.883,416.604,177.588,20.827,152.968
C03146=1093.106,304.635,416.636,177.585,20.824,152.967
C03147=1093.101,304.387,416.666,177.582,20.821,152.967
C03148=1093.096,304.139,416.697,177.578,20.818,152.967
C03149=1093.090,303.891,416.727,177.575,20.815,152.967
C03150=1093.081,303.500,416.776,177.571,20.811,152.967
C03151=1093.072,303.109,416.825,177.566,20.806,152.966
C03152=1093.063,302.719,416.873,177.561,20.801,152.966
C03153=1093.054,302.328,416.922,177.556,20.796,152.966
C03154=1093.049,302.079,416.953,177.553,20.793,152.966
C03155=1093.043,301.832,416.983,177.550,20.791,152.966
C03156=1093.037,301.584,417.014,177.547,20.788,152.965
C03157=1093.032,301.336,417.045,177.544,20.785,152.965
C03158=1093.026,301.088,417.075,177.541,20.782,152.965
C03159=1093.020,300.839,417.106,177.538,20.779,152.965
C03160=1093.015,300.591,417.137,177.534,20.777,152.965
C03161=1093.009,300.343,417.167,177.532,20.774,152.965
C03162=1093.004,300.095,417.198,177.529,20.771,152.964
C03163=1092.998,299.847,417.228,177.526,20.768,152.964
C03164=1092.992,299.600,417.259,177.523,20.765,152.964
C03165=1092.987,299.351,417.289,177.519,20.762,152.964
C03166=1092.982,299.103,417.319,177.516,20.759,152.964
C03167=1092.976,298.855,417.350,177.513,20.756,152.964
C03168=1092.971,298.607,417.381,177.510,20.753,152.963
C03169=1092.965,298.359,417.411,177.506,20.750,152.963
C03170=1092.959,298.111,417.441,177.503,20.747,152.963
C03171=1092.954,297.863,417.472,177.501,20.744,152.963
C03172=1092.948,297.615,417.502,177.497,20.742,152.963
C03173=1092.943,297.367,417.532,177.494,20.739,152.963
C03174=1092.937,297.119,417.563,177.491,20.736,152.963
C03175=1092.930,296.871,417.593,177.488,20.733,152.963
C03176=1092.925,296.623,417.624,177.485,20.731,152.962
C03177=1092.920,296.374,417.654,177.482,20.728,152.962
C03178=1092.914,296.126,417.684,177.479,20.725,152.962
C03179=1092.908,295.878,417.715,177.476,20.723,152.962
C03180=1092.903,295.630,417.744,177.473,20.720,152.962
C03181=1092.897,295.382,417.775,177.470,20.717,152.962
C03182=1092.891,295.134,417.805,177.467,20.714,152.962
C03183=1092.885,294.886,417.835,177.464,20.712,152.962
C03184=1092.880,294.638,417.865,177.461,20.709,152.961
C03185=1092.874,294.390,417.895,177.457,20.706,152.961
C03186=1092.868,294.142,417.925,177.454,20.703,152.961
C03187=1092.863,293.894,417.955,177.451,20.701,152.961
C03188=1092.857,293.646,417.985,177.448,20.698,152.961
C03189=1092.851,293.398,418.015,177.445,20.695,152.961
C03190=1092.845,293.150,418.046,177.442,20.692,152.961
C03191=1092.840,292.901,418.075,177.439,20.690,152.961
C03192=1092.834,292.654,418.106,177.436,20.687,152.961
C03193=1092.829,292.405,418.135,177.433,20.684,152.960
C03194=1092.823,292.157,418.166,177.430,20.681,152.960
C03195=1092.817,291.909,418.195,177.427,20.679,152.960
C03196=1092.811,291.661,418.226,177.423,20.676,152.960
C03197=1092.806,291.413,418.255,177.420,20.673,152.960
C03198=1092.800,291.164,418.285,177.417,20.671,152.960
C03199=1092.795,290.916,418.315,177.414,20.668,152.960
C03200=1092.789,290.668,418.345,177.411,20.665,152.960
C03201=1092.783,290.421,418.374,177.408,20.663,152.960
C03202=1092.774,290.043,418.420,177.403,20.659,152.959
C03203=1092.766,289.666,418.465,177.399,20.655,152.959
C03204=1092.757,289.289,418.510,177.394,20.651,152.959
C03205=1092.749,288.912,418.555,177.389,20.647,152.959
C03206=1092.743,288.664,418.586,177.386,20.644,152.959
C03207=1092.737,288.416,418.615,177.383,20.642,152.959
C03208=1092.731,288.168,418.644,177.380,20.639,152.959
C03209=1092.726,287.919,418.674,177.377,20.636,152.959
C03210=1092.720,287.671,418.704,177.374,20.634,152.959
C03211=1092.714,287.424,418.733,177.371,20.631,152.959
C03212=1092.709,287.175,418.763,177.368,20.628,152.958
C03213=1092.703,286.927,418.792,177.364,20.626,152.958
C03214=1092.697,286.679,418.821,177.361,20.623,152.958
C03215=1092.692,286.430,418.851,177.358,20.620,152.958
C03216=1092.686,286.183,418.881,177.355,20.618,152.958
C03217=1092.680,285.934,418.911,177.352,20.615,152.958
C03218=1092.674,285.686,418.940,177.349,20.613,152.958
C03219=1092.669,285.438,418.969,177.346,20.610,152.958
C03220=1092.664,285.190,418.999,177.343,20.607,152.958
C03221=1092.657,284.942,419.028,177.339,20.605,152.958
C03222=1092.652,284.693,419.057,177.336,20.602,152.958
C03223=1092.646,284.445,419.087,177.333,20.599,152.958
C03224=1092.641,284.197,419.116,177.330,20.597,152.958
C03225=1092.635,283.949,419.145,177.327,20.594,152.958
C03226=1092.630,283.700,419.175,177.325,20.592,152.957
C03227=1092.623,283.452,419.204,177.322,20.589,152.957
C03228=1092.618,283.204,419.234,177.318,20.587,152.957
C03229=1092.613,282.956,419.263,177.315,20.584,152.957
C03230=1092.607,282.708,419.292,177.312,20.582,152.957
C03231=1092.601,282.460,419.322,177.309,20.579,152.957
C03232=1092.596,282.211,419.351,177.306,20.576,152.957
C03233=1092.590,281.964,419.380,177.303,20.574,152.957
C03234=1092.585,281.715,419.410,177.300,20.571,152.957
C03235=1092.578,281.467,419.439,177.297,20.568,152.957
C03236=1092.573,281.219,419.468,177.293,20.566,152.957
C03237=1092.568,280.970,419.497,177.290,20.563,152.957
C03238=1092.562,280.722,419.526,177.287,20.561,152.957
C03239=1092.556,280.474,419.555,177.285,20.559,152.956
C03240=1092.550,280.226,419.585,177.282,20.556,152.956
C03241=1092.545,279.978,419.613,177.278,20.554,152.956
C03242=1092.539,279.729,419.642,177.275,20.551,152.956
C03243=1092.533,279.481,419.671,177.272,20.548,152.956
C03244=1092.528,279.233,419.700,177.269,20.546,152.956
C03245=1092.522,278.985,419.729,177.266,20.543,152.956
C03246=1092.517,278.736,419.758,177.263,20.541,152.956
C03247=1092.510,278.488,419.787,177.259,20.538,152.956
C03248=1092.506,278.240,419.817,177.256,20.536,152.956
C03249=1092.500,277.991,419.845,177.254,20.534,152.956
C03250=1092.493,277.743,419.874,177.251,20.531,152.956
C03251=1092.488,277.496,419.903,177.248,20.529,152.956
C03252=1092.483,277.247,419.932,177.245,20.526,152.956
C03253=1092.477,276.998,419.961,177.241,20.523,152.956
C03254=1092.469,276.631,420.003,177.237,20.520,152.956
C03255=1092.460,276.264,420.046,177.233,20.516,152.956
C03256=1092.451,275.896,420.089,177.228,20.513,152.956
C03257=1092.444,275.528,420.132,177.223,20.509,152.955
C03258=1092.438,275.280,420.160,177.220,20.506,152.955
C03259=1092.432,275.032,420.189,177.217,20.504,152.955
C03260=1092.427,274.783,420.218,177.214,20.501,152.955
C03261=1092.421,274.536,420.247,177.211,20.499,152.955
C03262=1092.415,274.287,420.275,177.208,20.497,152.955
C03263=1092.409,274.038,420.303,177.205,20.494,152.955
C03264=1092.404,273.790,420.333,177.202,20.492,152.955
C03265=1092.398,273.542,420.361,177.199,20.489,152.955
C03266=1092.393,273.294,420.390,177.195,20.487,152.955
C03267=1092.387,273.045,420.418,177.192,20.484,152.955
C03268=1092.381,272.797,420.448,177.190,20.482,152.955
C03269=1092.376,272.549,420.475,177.187,20.480,152.955
C03270=1092.370,272.300,420.504,177.184,20.477,152.955
C03271=1092.364,272.053,420.532,177.180,20.475,152.955
C03272=1092.358,271.804,420.561,177.177,20.472,152.955
C03273=1092.352,271.555,420.589,177.174,20.470,152.955
C03274=1092.348,271.308,420.618,177.171,20.467,152.955
C03275=1092.342,271.059,420.647,177.169,20.465,152.955
C03276=1092.336,270.811,420.675,177.165,20.463,152.955
C03277=1092.330,270.562,420.703,177.162,20.460,152.955
C03278=1092.325,270.315,420.732,177.159,20.458,152.955
C03279=1092.319,270.066,420.760,177.156,20.455,152.955
C03280=1092.313,269.818,420.788,177.153,20.453,152.955
C03281=1092.308,269.569,420.817,177.150,20.451,152.954
C03282=1092.303,269.321,420.845,177.147,20.449,152.955
C03283=1092.297,269.073,420.874,177.144,20.446,152.955
C03284=1092.291,268.824,420.902,177.141,20.444,152.954
C03285=1092.285,268.576,420.930,177.137,20.441,152.954
C03286=1092.280,268.328,420.958,177.134,20.439,152.954
C03287=1092.274,268.079,420.986,177.132,20.437,152.954
C03288=1092.269,267.831,421.014,177.129,20.434,152.954
C03289=1092.263,267.582,421.043,177.126,20.432,152.954
C03290=1092.257,267.334,421.071,177.122,20.429,152.954
C03291=1092.251,267.085,421.099,177.119,20.427,152.954
C03292=1092.246,266.838,421.128,177.116,20.425,152.954
C03293=1092.240,266.589,421.156,177.114,20.423,152.954
C03294=1092.235,266.341,421.184,177.110,20.420,152.954
C03295=1092.229,266.092,421.212,177.107,20.417,152.954
C03296=1092.223,265.844,421.240,177.104,20.415,152.954
C03297=1092.217,265.596,421.269,177.101,20.412,152.954
C03298=1092.212,265.347,421.297,177.098,20.410,152.954
C03299=1092.207,265.099,421.324,177.095,20.408,152.954
C03300=1092.201,264.850,421.352,177.092,20.406,152.954
C03301=1092.195,264.602,421.379,177.089,20.403,152.954
C03302=1092.189,264.354,421.408,177.086,20.401,152.954
C03303=1092.184,264.105,421.436,177.083,20.399,152.954
C03304=1092.178,263.857,421.464,177.080,20.396,152.954
C03305=1092.172,263.609,421.492,177.077,20.394,152.954
C03306=1092.163,263.244,421.533,177.072,20.391,152.954
C03307=1092.155,262.879,421.574,177.068,20.388,152.954
C03308=1092.146,262.514,421.615,177.063,20.384,152.954
C03309=1092.138,262.150,421.656,177.059,20.381,152.954
C03310=1092.132,261.900,421.683,177.056,20.379,152.954
C03311=1092.127,261.652,421.711,177.053,20.376,152.954
C03312=1092.121,261.404,421.739,177.049,20.374,152.954
C03313=1092.115,261.156,421.766,177.047,20.372,152.954
C03314=1092.110,260.907,421.794,177.044,20.370,152.954
C03315=1092.104,260.658,421.822,177.040,20.367,152.954
C03316=1092.098,260.411,421.849,177.037,20.365,152.954
C03317=1092.092,260.162,421.877,177.035,20.363,152.954
C03318=1092.087,259.913,421.905,177.032,20.361,152.954
C03319=1092.080,259.666,421.932,177.028,20.358,152.954
C03320=1092.075,259.416,421.960,177.025,20.356,152.954
C03321=1092.069,259.168,421.988,177.023,20.354,152.954
C03322=1092.063,258.920,422.015,177.019,20.352,152.954
C03323=1092.058,258.671,422.043,177.016,20.349,152.954
C03324=1092.052,258.423,422.071,177.013,20.347,152.954
C03325=1092.047,258.175,422.097,177.010,20.344,152.954
C03326=1092.041,257.926,422.126,177.007,20.342,152.954
C03327=1092.035,257.678,422.152,177.004,20.340,152.954
C03328=1092.030,257.429,422.180,177.001,20.338,152.954
C03329=1092.024,257.181,422.208,176.998,20.335,152.954
C03330=1092.018,256.932,422.235,176.995,20.333,152.954
C03331=1092.013,256.684,422.263,176.992,20.331,152.954
C03332=1092.007,256.436,422.290,176.989,20.329,152.954
C03333=1092.001,256.187,422.318,176.986,20.326,152.954
C03334=1091.996,255.939,422.346,176.983,20.325,152.954
C03335=1091.990,255.690,422.372,176.980,20.322,152.954
C03336=1091.985,255.442,422.400,176.977,20.320,152.954
C03337=1091.978,255.193,422.427,176.974,20.317,152.954
C03338=1091.973,254.945,422.455,176.971,20.316,152.954
C03339=1091.967,254.697,422.482,176.968,20.313,152.954
C03340=1091.962,254.448,422.509,176.965,20.311,152.954
C03341=1091.955,254.200,422.537,176.962,20.309,152.954
C03342=1091.950,253.951,422.564,176.959,20.307,152.954
C03343=1091.945,253.703,422.591,176.956,20.304,152.954
C03344=1091.939,253.454,422.619,176.953,20.302,152.954
C03345=1091.934,253.206,422.645,176.950,20.300,152.954
C03346=1091.928,252.957,422.672,176.947,20.298,152.954
C03347=1091.923,252.709,422.701,176.944,20.295,152.954
C03348=1091.917,252.460,422.727,176.941,20.293,152.954
C03349=1091.911,252.212,422.754,176.938,20.291,152.954
C03350=1091.906,251.963,422.781,176.935,20.288,152.954
C03351=1091.900,251.715,422.808,176.932,20.286,152.954
C03352=1091.895,251.467,422.836,176.929,20.284,152.954
C03353=1091.888,251.218,422.863,176.926,20.282,152.954
C03354=1091.883,250.969,422.890,176.923,20.279,152.954
C03355=1091.878,250.721,422.917,176.920,20.277,152.954
C03356=1091.873,250.472,422.944,176.917,20.275,152.954
C03357=1091.867,250.224,422.971,176.914,20.273,152.954
C03358=1091.859,249.857,423.011,176.909,20.269,152.954
C03359=1091.850,249.488,423.051,176.905,20.266,152.954
C03360=1091.842,249.121,423.092,176.901,20.263,152.954
C03361=1091.835,248.753,423.131,176.896,20.259,152.954
C03362=1091.829,248.505,423.158,176.893,20.257,152.954
C03363=1091.823,248.256,423.185,176.891,20.255,152.954
C03364=1091.818,248.008,423.212,176.887,20.253,152.954
C03365=1091.812,247.759,423.239,176.884,20.250,152.954
C03366=1091.807,247.510,423.266,176.882,20.249,152.954
C03367=1091.801,247.262,423.293,176.879,20.246,152.954
C03368=1091.795,247.013,423.319,176.875,20.244,152.954
C03369=1091.789,246.765,423.346,176.872,20.242,152.954
C03370=1091.784,246.516,423.373,176.870,20.240,152.954
C03371=1091.778,246.268,423.400,176.867,20.237,152.954
C03372=1091.773,246.019,423.427,176.863,20.235,152.955
C03373=1091.767,245.770,423.453,176.861,20.233,152.954
C03374=1091.762,245.522,423.480,176.857,20.231,152.955
C03375=1091.756,245.273,423.506,176.854,20.228,152.955
C03376=1091.751,245.025,423.533,176.852,20.226,152.954
C03377=1091.745,244.777,423.560,176.849,20.224,152.955
C03378=1091.739,244.528,423.586,176.845,20.222,152.955
C03379=1091.734,244.280,423.614,176.843,20.220,152.955
C03380=1091.729,244.031,423.640,176.840,20.218,152.955
C03381=1091.723,243.782,423.666,176.837,20.215,152.955
C03382=1091.717,243.534,423.693,176.834,20.213,152.955
C03383=1091.711,243.286,423.720,176.831,20.211,152.955
C03384=1091.706,243.037,423.747,176.828,20.209,152.955
C03385=1091.701,242.788,423.773,176.825,20.207,152.955
C03386=1091.695,242.540,423.799,176.822,20.205,152.955
C03387=1091.689,242.291,423.826,176.819,20.202,152.955
C03388=1091.684,242.042,423.852,176.816,20.201,152.955
C03389=1091.678,241.794,423.879,176.813,20.198,152.955
C03390=1091.672,241.546,423.905,176.810,20.196,152.955
C03391=1091.666,241.297,423.932,176.807,20.194,152.955
C03392=1091.661,241.048,423.958,176.804,20.192,152.955
C03393=1091.655,240.800,423.984,176.801,20.189,152.955
C03394=1091.650,240.551,424.010,176.798,20.188,152.955
C03395=1091.644,240.303,424.037,176.795,20.185,152.955
C03396=1091.638,240.054,424.064,176.793,20.183,152.955
C03397=1091.633,239.805,424.090,176.789,20.181,152.955
C03398=1091.627,239.557,424.116,176.786,20.179,152.955
C03399=1091.621,239.308,424.142,176.784,20.177,152.955
C03400=1091.616,239.059,424.169,176.780,20.175,152.955
C03401=1091.609,238.811,424.194,176.777,20.173,152.955
C03402=1091.604,238.562,424.221,176.775,20.171,152.955
C03403=1091.598,238.314,424.247,176.771,20.169,152.955
C03404=1091.593,238.066,424.273,176.769,20.167,152.955
C03405=1091.587,237.817,424.300,176.766,20.164,152.955
C03406=1091.582,237.568,424.326,176.762,20.162,152.955
C03407=1091.576,237.320,424.352,176.760,20.160,152.955
C03408=1091.571,237.071,424.378,176.757,20.158,152.955
C03409=1091.565,236.822,424.404,176.754,20.155,152.955
C03410=1091.556,236.448,424.443,176.750,20.152,152.955
C03411=1091.548,236.073,424.483,176.745,20.149,152.956
C03412=1091.540,235.699,424.522,176.741,20.146,152.956
C03413=1091.532,235.324,424.562,176.736,20.143,152.956
C03414=1091.525,235.075,424.587,176.733,20.141,152.956
C03415=1091.520,234.826,424.613,176.730,20.139,152.956
C03416=1091.514,234.578,424.640,176.728,20.137,152.956
C03417=1091.509,234.329,424.666,176.724,20.135,152.956
C03418=1091.503,234.080,424.691,176.722,20.133,152.956
C03419=1091.497,233.833,424.717,176.719,20.130,152.956
C03420=1091.492,233.584,424.743,176.715,20.128,152.956
C03421=1091.486,233.335,424.769,176.713,20.126,152.956
C03422=1091.481,233.086,424.795,176.710,20.124,152.956
C03423=1091.474,232.838,424.821,176.707,20.122,152.956
C03424=1091.470,232.590,424.847,176.704,20.120,152.956
C03425=1091.464,232.341,424.873,176.701,20.117,152.956
C03426=1091.459,232.092,424.898,176.698,20.116,152.956
C03427=1091.452,231.843,424.924,176.695,20.113,152.956
C03428=1091.447,231.595,424.950,176.693,20.112,152.956
C03429=1091.442,231.346,424.976,176.689,20.109,152.956
C03430=1091.436,231.097,425.002,176.686,20.107,152.956
C03431=1091.430,230.849,425.027,176.684,20.105,152.956
C03432=1091.425,230.600,425.053,176.681,20.103,152.956
C03433=1091.420,230.351,425.079,176.678,20.101,152.956
C03434=1091.414,230.103,425.104,176.675,20.099,152.956
C03435=1091.408,229.854,425.130,176.672,20.097,152.956
C03436=1091.402,229.605,425.155,176.669,20.095,152.957
C03437=1091.397,229.357,425.181,176.666,20.093,152.957
C03438=1091.391,229.108,425.206,176.663,20.091,152.957
C03439=1091.385,228.860,425.233,176.660,20.089,152.957
C03440=1091.379,228.611,425.258,176.657,20.087,152.957
C03441=1091.374,228.363,425.284,176.654,20.085,152.957
C03442=1091.368,228.114,425.309,176.652,20.083,152.957
C03443=1091.362,227.865,425.335,176.649,20.080,152.957
C03444=1091.357,227.616,425.360,176.645,20.078,152.957
C03445=1091.352,227.368,425.385,176.643,20.076,152.957
C03446=1091.346,227.119,425.411,176.639,20.074,152.957
C03447=1091.340,226.870,425.437,176.637,20.072,152.957
C03448=1091.335,226.622,425.462,176.634,20.070,152.957
C03449=1091.329,226.373,425.487,176.631,20.069,152.957
C03450=1091.323,226.124,425.513,176.628,20.066,152.957
C03451=1091.318,225.876,425.538,176.626,20.065,152.957
C03452=1091.312,225.627,425.564,176.622,20.062,152.957
C03453=1091.306,225.378,425.590,176.619,20.060,152.957
C03454=1091.301,225.130,425.614,176.617,20.058,152.957
C03455=1091.295,224.881,425.640,176.613,20.056,152.957
C03456=1091.289,224.632,425.665,176.611,20.054,152.957
C03457=1091.284,224.384,425.691,176.608,20.052,152.958
C03458=1091.278,224.135,425.716,176.605,20.050,152.957
C03459=1091.273,223.886,425.741,176.602,20.048,152.958
C03460=1091.267,223.638,425.766,176.600,20.046,152.958
C03461=1091.261,223.389,425.792,176.596,20.044,152.958
C03462=1091.253,223.006,425.831,176.592,20.041,152.958
C03463=1091.244,222.623,425.870,176.587,20.037,152.958
C03464=1091.236,222.239,425.908,176.583,20.034,152.958
C03465=1091.228,221.856,425.947,176.578,20.031,152.958
C03466=1091.222,221.607,425.972,176.576,20.029,152.958
C03467=1091.216,221.358,425.997,176.573,20.027,152.958
C03468=1091.210,221.110,426.022,176.570,20.025,152.958
C03469=1091.205,220.861,426.048,176.567,20.023,152.958
C03470=1091.199,220.613,426.073,176.565,20.021,152.958
C03471=1091.193,220.363,426.097,176.561,20.019,152.958
C03472=1091.187,220.115,426.123,176.559,20.017,152.958
C03473=1091.182,219.867,426.148,176.555,20.015,152.958
C03474=1091.176,219.617,426.173,176.553,20.013,152.958
C03475=1091.171,219.369,426.198,176.550,20.011,152.958
C03476=1091.165,219.120,426.222,176.547,20.009,152.959
C03477=1091.159,218.872,426.247,176.544,20.007,152.959
C03478=1091.154,218.622,426.272,176.541,20.005,152.959
C03479=1091.148,218.374,426.297,176.538,20.003,152.959
C03480=1091.143,218.125,426.322,176.536,20.001,152.959
C03481=1091.137,217.877,426.347,176.532,19.999,152.959
C03482=1091.131,217.628,426.372,176.530,19.997,152.959
C03483=1091.126,217.380,426.397,176.527,19.995,152.959
C03484=1091.120,217.130,426.422,176.524,19.993,152.959
C03485=1091.115,216.882,426.446,176.521,19.991,152.959
C03486=1091.109,216.633,426.471,176.519,19.989,152.959
C03487=1091.104,216.385,426.496,176.515,19.987,152.959
C03488=1091.097,216.136,426.521,176.513,19.985,152.959
C03489=1091.092,215.887,426.545,176.510,19.983,152.959
C03490=1091.087,215.638,426.571,176.507,19.981,152.959
C03491=1091.081,215.390,426.595,176.504,19.979,152.959
C03492=1091.075,215.140,426.620,176.502,19.977,152.959
C03493=1091.070,214.892,426.644,176.498,19.975,152.959
C03494=1091.064,214.644,426.669,176.496,19.973,152.959
C03495=1091.059,214.395,426.694,176.493,19.971,152.959
C03496=1091.053,214.146,426.718,176.490,19.969,152.960
C03497=1091.047,213.897,426.744,176.487,19.967,152.960
C03498=1091.042,213.648,426.768,176.484,19.965,152.960
C03499=1091.037,213.399,426.793,176.482,19.963,152.960
C03500=1091.031,213.151,426.817,176.479,19.961,152.960
C03501=1091.026,212.903,426.842,176.476,19.959,152.960
C03502=1091.020,212.653,426.867,176.473,19.957,152.960
C03503=1091.014,212.405,426.891,176.471,19.955,152.960
C03504=1091.009,212.155,426.916,176.467,19.953,152.960
C03505=1091.003,211.907,426.940,176.465,19.951,152.960
C03506=1090.997,211.659,426.964,176.461,19.949,152.960
C03507=1090.991,211.410,426.989,176.459,19.947,152.960
C03508=1090.986,211.161,427.013,176.456,19.945,152.960
C03509=1090.980,210.913,427.038,176.453,19.943,152.960
C03510=1090.975,210.663,427.062,176.450,19.941,152.960
C03511=1090.969,210.415,427.086,176.448,19.939,152.960
C03512=1090.963,210.165,427.111,176.445,19.937,152.960
C03513=1090.958,209.917,427.135,176.442,19.935,152.960
C03514=1090.949,209.538,427.173,176.438,19.932,152.960
C03515=1090.940,209.158,427.210,176.434,19.930,152.961
C03516=1090.933,208.779,427.247,176.429,19.926,152.961
C03517=1090.924,208.400,427.284,176.425,19.923,152.961
C03518=1090.900,207.379,427.383,176.359,19.891,152.965
C03519=1090.895,207.129,427.406,176.356,19.890,152.965
C03520=1090.889,206.881,427.430,176.354,19.889,152.966
C03521=1090.884,206.632,427.454,176.351,19.888,152.966
C03522=1090.879,206.383,427.478,176.347,19.887,152.966
C03523=1090.872,206.134,427.502,176.344,19.886,152.966
C03524=1090.867,205.886,427.526,176.341,19.885,152.967
C03525=1090.861,205.637,427.550,176.339,19.884,152.967
C03526=1090.856,205.388,427.573,176.336,19.883,152.967
C03527=1090.851,205.140,427.597,176.333,19.882,152.967
C03528=1090.845,204.891,427.620,176.330,19.881,152.968
C03529=1090.839,204.641,427.645,176.327,19.879,152.968
C03530=1090.833,204.393,427.669,176.324,19.878,152.968
C03531=1090.828,204.144,427.692,176.321,19.877,152.969
C03532=1090.823,203.895,427.717,176.318,19.877,152.969
C03533=1090.817,203.646,427.739,176.315,19.876,152.969
C03534=1090.812,203.398,427.764,176.313,19.875,152.969
C03535=1090.806,203.150,427.787,176.309,19.873,152.970
C03536=1090.801,202.900,427.811,176.306,19.872,152.970
C03537=1090.794,202.651,427.835,176.303,19.871,152.970
C03538=1090.789,202.402,427.858,176.301,19.870,152.970
C03539=1090.783,202.154,427.882,176.298,19.869,152.971
C03540=1090.778,201.905,427.906,176.295,19.868,152.971
C03541=1090.772,201.656,427.929,176.292,19.867,152.971
C03542=1090.766,201.408,427.952,176.288,19.866,152.972
C03543=1090.760,201.158,427.977,176.286,19.865,152.972
C03544=1090.755,200.909,428.000,176.283,19.863,152.972
C03545=1090.749,200.661,428.024,176.280,19.862,152.972
C03546=1090.744,200.412,428.047,176.277,19.862,152.973
C03547=1090.738,200.163,428.070,176.274,19.861,152.973
C03548=1090.733,199.914,428.094,176.272,19.860,152.973
C03549=1090.727,199.666,428.117,176.269,19.859,152.973
C03550=1090.721,199.417,428.141,176.265,19.857,152.974
C03551=1090.716,199.168,428.164,176.262,19.856,152.974
C03552=1090.710,198.918,428.188,176.260,19.855,152.974
C03553=1090.703,198.670,428.211,176.257,19.854,152.975
C03554=1090.698,198.421,428.235,176.254,19.853,152.975
C03555=1090.693,198.172,428.258,176.251,19.852,152.975
C03556=1090.687,197.924,428.282,176.248,19.851,152.975
C03557=1090.681,197.675,428.304,176.245,19.850,152.976
C03558=1090.676,197.426,428.328,176.243,19.849,152.976
C03559=1090.670,197.177,428.352,176.240,19.848,152.976
C03560=1090.664,196.928,428.375,176.236,19.847,152.976
C03561=1090.659,196.679,428.398,176.234,19.846,152.977
C03562=1090.653,196.430,428.421,176.231,19.845,152.977
C03563=1090.647,196.182,428.445,176.228,19.843,152.977
C03564=1090.642,195.933,428.468,176.225,19.842,152.977
C03565=1090.637,195.684,428.491,176.222,19.842,152.978
C03566=1090.631,195.435,428.514,176.219,19.841,152.978
C03567=1090.625,195.186,428.537,176.217,19.840,152.978
C03568=1090.620,194.938,428.561,176.214,19.839,152.979
C03569=1090.614,194.689,428.584,176.211,19.838,152.979
C03570=1090.609,194.440,428.607,176.207,19.836,152.979
C03571=1090.603,194.191,428.630,176.205,19.835,152.979
C03572=1090.598,193.942,428.654,176.202,19.834,152.980
C03573=1090.592,193.693,428.677,176.199,19.833,152.980
C03574=1090.586,193.444,428.700,176.196,19.832,152.980
C03575=1090.580,193.196,428.723,176.194,19.831,152.980
C03576=1090.575,192.947,428.746,176.191,19.830,152.981
C03577=1090.570,192.698,428.770,176.188,19.829,152.981
C03578=1090.564,192.449,428.793,176.185,19.828,152.981
C03579=1090.558,192.172,428.818,176.182,19.826,152.981
C03580=1090.552,191.895,428.844,176.179,19.825,152.982
C03581=1090.546,191.620,428.869,176.176,19.824,152.982
C03582=1090.540,191.342,428.894,176.172,19.823,152.982
C03583=1090.534,191.094,428.917,176.170,19.822,152.983
C03584=1090.528,190.845,428.940,176.167,19.820,152.983
C03585=1090.523,190.595,428.964,176.164,19.819,152.983
C03586=1090.518,190.347,428.987,176.161,19.818,152.983
C03587=1090.512,190.098,429.010,176.159,19.817,152.984
C03588=1090.506,189.849,429.033,176.156,19.816,152.984
C03589=1090.500,189.600,429.056,176.153,19.815,152.984
C03590=1090.495,189.352,429.078,176.150,19.814,152.984
C03591=1090.490,189.103,429.101,176.147,19.813,152.985
C03592=1090.485,188.854,429.125,176.145,19.812,152.985
C03593=1090.479,188.605,429.148,176.142,19.811,152.985
C03594=1090.473,188.356,429.171,176.139,19.809,152.985
C03595=1090.467,188.107,429.194,176.136,19.808,152.985
C03596=1090.462,187.859,429.216,176.133,19.807,152.986
C03597=1090.457,187.609,429.238,176.130,19.806,152.986
C03598=1090.451,187.360,429.261,176.127,19.805,152.986
C03599=1090.446,187.111,429.285,176.125,19.804,152.986
C03600=1090.440,186.862,429.308,176.122,19.802,152.987
C03601=1090.435,186.614,429.330,176.119,19.801,152.987
C03602=1090.430,186.365,429.353,176.117,19.800,152.987
C03603=1090.424,186.116,429.376,176.114,19.799,152.987
C03604=1090.418,185.867,429.398,176.111,19.798,152.988
C03605=1090.413,185.618,429.421,176.108,19.797,152.988
C03606=1090.408,185.370,429.444,176.105,19.796,152.988
C03607=1090.402,185.120,429.466,176.103,19.794,152.988
C03608=1090.396,184.871,429.489,176.100,19.793,152.988
C03609=1090.391,184.622,429.512,176.097,19.792,152.989
C03610=1090.385,184.373,429.535,176.095,19.791,152.989
C03611=1090.379,184.125,429.556,176.092,19.791,152.989
C03612=1090.374,183.876,429.579,176.089,19.790,152.990
C03613=1090.368,183.627,429.602,176.086,19.789,152.990
C03614=1090.362,183.378,429.624,176.083,19.788,152.990
C03615=1090.356,183.129,429.647,176.081,19.787,152.990
C03616=1090.350,182.880,429.670,176.078,19.786,152.991
C03617=1090.345,182.631,429.692,176.075,19.785,152.991
C03618=1090.340,182.382,429.715,176.072,19.783,152.991
C03619=1090.333,182.134,429.737,176.069,19.782,152.991
C03620=1090.328,181.884,429.759,176.067,19.781,152.992
C03621=1090.322,181.635,429.782,176.064,19.780,152.992
C03622=1090.317,181.386,429.804,176.061,19.779,152.992
C03623=1090.311,181.138,429.826,176.059,19.778,152.992
C03624=1090.305,180.888,429.849,176.056,19.777,152.993
C03625=1090.300,180.640,429.872,176.053,19.776,152.993
C03626=1090.293,180.391,429.894,176.050,19.775,152.993
C03627=1090.288,180.141,429.916,176.047,19.774,152.993
C03628=1090.283,179.893,429.939,176.045,19.773,152.994
C03629=1090.276,179.644,429.960,176.042,19.772,152.994
C03630=1090.271,179.395,429.983,176.039,19.771,152.994
C03631=1090.265,179.146,430.005,176.036,19.769,152.994
